# B&R Automation Studio project NAEUL004C00R13L518F00 (part 76)

#### Act_Main.st
```iecst
(** 2019-05-28 **)
ACTION Act_Main:

	IF eStatOld <> eStat THEN
		fbInit(bEn := FALSE);
		fbEnt(bEn := FALSE);
		fbPreExit(bEn := FALSE);
		fbExit(bEn := FALSE);
		fbExit1(bEn := FALSE);
		fbStop(bEn := FALSE);
		fbClprClampChk(bEn := FALSE);
		fbClprUnclampChk(bEn := FALSE);

		IF eStatOld <> MagConvActIdle
			AND eStatOld <> MagConvActSetMtrSigOnOrLToR
			AND eStatOld <> MagConvActSetMtrDirOrRToL
			AND eStatOld <> MagConvActRstMtrSigOnOrLToR
			AND eStatOld <> MagConvActRstMtrDirOrRToL
			AND eStatOld <> MagConvActSetMtrAll
			AND eStatOld <> MagConvActRstMtrAll THEN

			bMtrSigOnOrLToR	:= FALSE;
			bMtrDirOrRToL	:= FALSE;

		END_IF

		usiStep		:= 0;
		bReachEnd	:= FALSE;

		sStatTxt	:= a_sStatText[eStat];

		eStatOld	:= eStat;

		eStatus		:= Busy;
	END_IF

	//Main
	CASE eStat OF

		MagConvActIdle:
			IF EDGENEG(p_bManual) THEN
				bMtrSigOnOrLToR	:= FALSE;
				bMtrDirOrRToL	:= FALSE;
			END_IF

			eStatus	:= Idle;

		MagConvActInit:
			IF eStatus = Idle OR eStatus = Busy THEN

				eStatus	:= Busy;

				//Magazine Conveyor Init Run
				//Detect Have Magazine
				IF p_bLeftSen OR p_bRightSen THEN
					bHvMag	:= TRUE;
				ELSE
					bHvMag	:= FALSE;
				END_IF

				fbInit.bConvLToR	:= (p_eDirection = ConvDirLToR) OR (p_eDirection = ConvDirLToL);
				fbInit.tTxDlyTm		:= DINT_TO_TIME(p_diInitTm);

				IF fbInit.bConvLToR = TRUE THEN
					fbInit.bEndSen	:= p_bRightSen;
				ELSE
					fbInit.bEndSen	:= p_bLeftSen;
				END_IF

				fbInit(bEn := TRUE);

				bMtrSigOnOrLToR	:= fbInit.bMtrSigOnOrLToR;
				bMtrDirOrRToL	:= fbInit.bMtrDirOrRToL;

				IF fbInit.udiStatus = 0 THEN
					IF fbInit.bConvLToR = TRUE THEN
						IF bHvMag = TRUE AND p_bRightSen = FALSE THEN
							udiStatus	:= 10000;	//Magazine Detected But Not Present At Outlet Sensor (L - R) While Magazine Conveyor Initial
							eStatus		:= Error;
						ELSE
							eStatus	:= Done;
						END_IF
					ELSE
						IF bHvMag = TRUE AND p_bLeftSen = FALSE THEN
							udiStatus	:= 10001;	//Magazine Detected But Not Present At Outlet Sensor (R - L) While Magazine Conveyor Initial
							eStatus		:= Error;
						ELSE
							eStatus	:= Done;
						END_IF
					END_IF
				ELSIF fbInit.udiStatus < 65534 THEN
					udiStatus	:= fbInit.udiStatus;
					eStatus		:= Error;
				END_IF
			END_IF

		MagConvActInitStopClp:
			IF eStatus = Idle OR eStatus = Busy THEN

				eStatus	:= Busy;

				CASE usiStep OF
					0: //Unclamp
						bClprClampCtrl		:= FALSE;

						fbClprUnclampChk.bExtSen	:= p_bClprClampSen;
						fbClprUnclampChk.bRetSen	:= p_bClprUnclampSen;
						fbClprUnclampChk.bRetSafety	:= p_bClprUnclampSafetySen;
						fbClprUnclampChk(bEn := TRUE);

						IF fbClprUnclampChk.udiStatus = 0 THEN
							usiStep	:= 1;
						ELSIF fbClprUnclampChk.udiStatus < 65534 THEN
							bClprClampCtrl		:= TRUE;

							eStatus			:= Error;

							IF fbClprUnclampChk.udiStatus = 1504 THEN
								udiStatus	:= 10002;	//Clamper Clamp Sensor Off Time Out In Unclamp Check While Conveyor Initial With Clamper
							ELSIF fbClprUnclampChk.udiStatus = 1505 THEN
								udiStatus	:= 10003;	//Clamper Unclamp Sensor On Time Out In Unclamp Check While Conveyor Initial With Clamper
							ELSIF fbClprUnclampChk.udiStatus = 1508 THEN
								udiStatus	:= 10004;	//Clamper Unclamp Safety Sensor Error In Unclamp Check While Conveyor Initial With Clamper
							ELSE
								udiStatus	:= fbClprUnclampChk.udiStatus;
							END_IF
						END_IF

					1:	//Magazine Conveyor Init Run
						//Detect Have Magazine
						IF p_bLeftSen OR p_bRightSen THEN
							bHvMag	:= TRUE;
						ELSE
							bHvMag	:= FALSE;
						END_IF

						fbInit.bConvLToR	:= (p_eDirection = ConvDirLToR) OR (p_eDirection = ConvDirLToL);
						fbInit.tTxDlyTm		:= DINT_TO_TIME(p_diInitTm);

						IF fbInit.bConvLToR = TRUE THEN
							fbInit.bEndSen	:= p_bRightSen;
						ELSE
							fbInit.bEndSen	:= p_bLeftSen;
						END_IF

						fbInit(bEn := TRUE);

						bMtrSigOnOrLToR	:= fbInit.bMtrSigOnOrLToR;
						bMtrDirOrRToL	:= fbInit.bMtrDirOrRToL;

						IF fbInit.udiStatus = 0 THEN
							IF fbInit.bConvLToR = TRUE THEN
								IF bHvMag = TRUE AND p_bRightSen = FALSE THEN
									udiStatus	:= 10005;	//Magazine Detected But Not Present At Outlet Sensor (L - R) While Conveyor Initial With Clamper
									eStatus		:= Error;
								ELSE
									usiStep	:= 2;
								END_IF
							ELSE
								IF bHvMag = TRUE AND p_bLeftSen = FALSE THEN
									udiStatus	:= 10006;	//Magazine Detected But Not Present At Outlet Sensor (R - L) While Conveyor Initial With Clamper
									eStatus		:= Error;
								ELSE
									usiStep	:= 2;
								END_IF
							END_IF
						ELSIF fbInit.udiStatus < 65534 THEN
							udiStatus	:= fbInit.udiStatus;
							eStatus		:= Error;
						END_IF

					2:	//Check If Have Magazine
						IF bHvMag = TRUE THEN
							usiStep	:= 3;
						ELSE
							eStatus	:= Done;
						END_IF

					3:	//Clamp
						bClprClampCtrl		:= TRUE;

						fbClprClampChk.bExtSen		:= p_bClprClampSen;
						fbClprClampChk.bRetSen		:= p_bClprUnclampSen;
						fbClprClampChk.bExtSafety	:= p_bClprClampSafetySen;
						fbClprClampChk(bEn := TRUE);

						IF fbClprClampChk.udiStatus = 0 THEN
							eStatus		:= Done;
						ELSIF fbClprClampChk.udiStatus < 65534 THEN
							bClprClampCtrl		:= FALSE;

							eStatus			:= Error;

							IF fbClprClampChk.udiStatus = 1503 THEN
								udiStatus	:= 10007;	//Clamper Clamp Sensor On Time Out In Clamp Check While Conveyor Initial With Clamper
							ELSIF fbClprClampChk.udiStatus = 1506 THEN
								udiStatus	:= 10008;	//Clamper Unclamp Sensor Off Time Out In Clamp Check While Conveyor Initial With Clamper
							ELSIF fbClprClampChk.udiStatus = 1507 THEN
								udiStatus	:= 10009;	//Clamper Clamp Safety Sensor Error In Clamp Check While Conveyor Initial With Clamper
							ELSE
								udiStatus	:= fbClprClampChk.udiStatus;
							END_IF
						END_IF

				END_CASE
			END_IF

		MagConvActInitClpStop:
			IF eStatus = Idle OR eStatus = Busy THEN

				eStatus	:= Busy;

				CASE usiStep OF
					0: //Unclamp
						bClprClampCtrl		:= FALSE;

						fbClprUnclampChk.bExtSen	:= p_bClprClampSen;
						fbClprUnclampChk.bRetSen	:= p_bClprUnclampSen;
						fbClprUnclampChk.bRetSafety	:= p_bClprUnclampSafetySen;
						fbClprUnclampChk(bEn := TRUE);

						IF fbClprUnclampChk.udiStatus = 0 THEN
							usiStep	:= 1;
						ELSIF fbClprUnclampChk.udiStatus < 65534 THEN
							bClprClampCtrl		:= TRUE;

							eStatus			:= Error;

							IF fbClprUnclampChk.udiStatus = 1504 THEN
								udiStatus	:= 10038;	//Clamper Clamp Sensor Off Time Out In Unclamp Check While Conveyor Initial With Clamper
							ELSIF fbClprUnclampChk.udiStatus = 1505 THEN
								udiStatus	:= 10039;	//Clamper Unclamp Sensor On Time Out In Unclamp Check While Conveyor Initial With Clamper
							ELSIF fbClprUnclampChk.udiStatus = 1508 THEN
								udiStatus	:= 10040;	//Clamper Unclamp Safety Sensor Error In Unclamp Check While Conveyor Initial With Clamper
							ELSE
								udiStatus	:= fbClprUnclampChk.udiStatus;
							END_IF
						END_IF

					1:	//Magazine Conveyor Init Run & Clamp
						//Detect Have Magazine
						IF p_bLeftSen OR p_bRightSen THEN
							bHvMag	:= TRUE;
						ELSE
							bHvMag	:= FALSE;
						END_IF

						fbInit.bConvLToR	:= (p_eDirection = ConvDirLToR) OR (p_eDirection = ConvDirLToL);
						fbInit.tTxDlyTm		:= DINT_TO_TIME(p_diInitTm);

						IF fbInit.bConvLToR = TRUE THEN
							fbInit.bEndSen	:= p_bRightSen;
						ELSE
							fbInit.bEndSen	:= p_bLeftSen;
						END_IF

						fbInit(bEn := TRUE);

						bMtrSigOnOrLToR	:= fbInit.bMtrSigOnOrLToR;
						bMtrDirOrRToL	:= fbInit.bMtrDirOrRToL;

						IF fbInit.bEndSen = TRUE THEN
							bReachEnd	:= TRUE;
						END_IF

						IF bReachEnd = TRUE THEN
							fbClprDlyTm(IN := TRUE);

							IF fbClprDlyTm.Q = TRUE THEN
								bClprClampCtrl		:= TRUE;

								fbClprClampChk.bExtSen		:= p_bClprClampSen;
								fbClprClampChk.bRetSen		:= p_bClprUnclampSen;
								fbClprClampChk.bExtSafety	:= p_bClprClampSafetySen;
								fbClprClampChk(bEn := TRUE);
							END_IF

						END_IF

						IF (fbInit.udiStatus = 0) AND ((fbClprClampChk.udiStatus = 0) OR (bReachEnd = FALSE)) THEN
							IF fbInit.bConvLToR = TRUE THEN
								IF bHvMag = TRUE AND p_bRightSen = FALSE THEN
									udiStatus	:= 10041;	//Magazine Detected But Not Present At Outlet Sensor (L - R) While Conveyor Initial With Clamper
									eStatus		:= Error;
								ELSE
									eStatus		:= Done;
								END_IF
							ELSE
								IF bHvMag = TRUE AND p_bLeftSen = FALSE THEN
									udiStatus	:= 10042;	//Magazine Detected But Not Present At Outlet Sensor (R - L) While Conveyor Initial With Clamper
									eStatus		:= Error;
								ELSE
									eStatus		:= Done;
								END_IF
							END_IF

						ELSIF fbInit.udiStatus > 0 AND fbInit.udiStatus < 65534 THEN
							udiStatus	:= fbInit.udiStatus;
							eStatus		:= Error;

						ELSIF fbClprClampChk.udiStatus > 0 AND fbClprClampChk.udiStatus < 65534 THEN
							bClprClampCtrl		:= FALSE;

							eStatus			:= Error;

							IF fbClprClampChk.udiStatus = 1503 THEN
								udiStatus	:= 10043;	//Clamper Clamp Sensor On Time Out In Clamp Check While Conveyor Initial With Clamper
							ELSIF fbClprClampChk.udiStatus = 1506 THEN
								udiStatus	:= 10044;	//Clamper Unclamp Sensor Off Time Out In Clamp Check While Conveyor Initial With Clamper
							ELSIF fbClprClampChk.udiStatus = 1507 THEN
								udiStatus	:= 10045;	//Clamper Clamp Safety Sensor Error In Clamp Check While Conveyor Initial With Clamper
							ELSE
								udiStatus	:= fbClprClampChk.udiStatus;
							END_IF
						END_IF

				END_CASE
			END_IF

		MagConvActEnt:
			IF eStatus = Idle OR eStatus = Busy THEN

				eStatus	:= Busy;

				//Detect Have Magazine
				IF p_bLeftSen OR p_bRightSen THEN
					bHvMag	:= TRUE;
				END_IF

				//Conveyor Run
				fbEnt.bConvLToR		:= (p_eDirection = ConvDirLToR) OR (p_eDirection = ConvDirLToL);
				fbEnt.tTimeOut		:= DINT_TO_TIME(p_diTxInTimeOut);

				IF fbEnt.bConvLToR = TRUE THEN
					fbEnt.bEndSen	:= p_bRightSen;
				ELSE
					fbEnt.bEndSen	:= p_bLeftSen;
				END_IF

				fbEnt(bEn := TRUE);

				bMtrSigOnOrLToR	:= fbEnt.bMtrSigOnOrLToR;
				bMtrDirOrRToL	:= fbEnt.bMtrDirOrRToL;

				IF fbEnt.udiStatus = 0 THEN
					eStatus		:= Done;
				ELSIF fbEnt.udiStatus < 65534 THEN
					eStatus		:= Error;

					IF fbEnt.udiStatus = 1101 THEN
						udiStatus	:= 10028;	//Transfer In Time Out While Entering Magazine
					ELSE
						udiStatus	:= fbEnt.udiStatus;
					END_IF
				END_IF

			END_IF

		MagConvActEntStopClp:
			IF eStatus = Idle OR eStatus = Busy THEN

				eStatus	:= Busy;

				CASE usiStep OF
					0:
						//Detect Have Magazine
						IF p_bLeftSen OR p_bRightSen THEN
							bHvMag	:= TRUE;
						END_IF

						//Conveyor Run
						fbEnt.bConvLToR		:= (p_eDirection = ConvDirLToR) OR (p_eDirection = ConvDirLToL);
						fbEnt.tTimeOut		:= DINT_TO_TIME(p_diTxInTimeOut);

						IF fbEnt.bConvLToR = TRUE THEN
							fbEnt.bEndSen	:= p_bRightSen;
						ELSE
							fbEnt.bEndSen	:= p_bLeftSen;
						END_IF

						fbEnt(bEn := TRUE);

						bMtrSigOnOrLToR	:= fbEnt.bMtrSigOnOrLToR;
						bMtrDirOrRToL	:= fbEnt.bMtrDirOrRToL;

						IF fbEnt.udiStatus = 0 THEN
							usiStep	:= 1;
						ELSIF fbEnt.udiStatus < 65534 THEN
							eStatus		:= Error;

							IF fbEnt.udiStatus = 1101 THEN
								udiStatus	:= 10029;	//Transfer In Time Out While Entering Magazine
							ELSE
								udiStatus	:= fbEnt.udiStatus;
							END_IF
						END_IF

					1:
						bClprClampCtrl		:= TRUE;

						fbClprClampChk.bExtSen		:= p_bClprClampSen;
						fbClprClampChk.bRetSen		:= p_bClprUnclampSen;
						fbClprClampChk.bExtSafety	:= p_bClprClampSafetySen;
						fbClprClampChk(bEn := TRUE);

						IF fbClprClampChk.udiStatus = 0 THEN
							eStatus		:= Done;
						ELSIF fbClprClampChk.udiStatus < 65534 THEN
							bClprClampCtrl		:= FALSE;

							eStatus			:= Error;

							IF fbClprClampChk.udiStatus = 1503 THEN
								udiStatus	:= 10010;	//Clamper Clamp Sensor On Time Out In Clamp Check While Conveyor Enter With Clamper
							ELSIF fbClprClampChk.udiStatus = 1506 THEN
								udiStatus	:= 10011;	//Clamper Unclamp Sensor Off Time Out In Clamp Check While Conveyor Enter With Clamper
							ELSIF fbClprClampChk.udiStatus = 1507 THEN
								udiStatus	:= 10012;	//Clamper Clamp Safety Sensor Error In Clamp Check While Conveyor Enter With Clamper
							ELSE
								udiStatus	:= fbClprClampChk.udiStatus;
							END_IF
						END_IF

				END_CASE

			END_IF

		MagConvActEntClpStop:
			IF eStatus = Idle OR eStatus = Busy THEN

				eStatus	:= Busy;

				//Detect Have Magazine
				IF p_bLeftSen OR p_bRightSen THEN
					bHvMag	:= TRUE;
				END_IF

				//Conveyor Run
				fbEnt.bConvLToR		:= (p_eDirection = ConvDirLToR) OR (p_eDirection = ConvDirLToL);
				fbEnt.tTimeOut		:= DINT_TO_TIME(p_diTxInTimeOut);

				IF fbEnt.bConvLToR = TRUE THEN
					fbEnt.bEndSen	:= p_bRightSen;
				ELSE
					fbEnt.bEndSen	:= p_bLeftSen;
				END_IF

				fbEnt(bEn := TRUE);

				bMtrSigOnOrLToR	:= fbEnt.bMtrSigOnOrLToR;
				bMtrDirOrRToL	:= fbEnt.bMtrDirOrRToL;

				IF fbEnt.bEndSen = TRUE THEN
					bReachEnd	:= TRUE;
				END_IF

				IF bReachEnd = TRUE THEN
					fbClprDlyTm(IN := TRUE);

					IF fbClprDlyTm.Q = TRUE THEN
						bClprClampCtrl		:= TRUE;

						fbClprClampChk.bExtSen		:= p_bClprClampSen;
						fbClprClampChk.bRetSen		:= p_bClprUnclampSen;
						fbClprClampChk.bExtSafety	:= p_bClprClampSafetySen;
						fbClprClampChk(bEn := TRUE);
					END_IF

				END_IF

				IF fbClprClampChk.udiStatus = 0 AND fbEnt.udiStatus = 0 THEN
					eStatus		:= Done;

				ELSIF fbClprClampChk.udiStatus > 0 AND fbClprClampChk.udiStatus < 65534 THEN
					bClprClampCtrl		:= FALSE;

					eStatus			:= Error;

					IF fbClprClampChk.udiStatus = 1503 THEN
						udiStatus	:= 10034;	//Clamper Clamp Sensor On Time Out In Clamp Check While Conveyor Enter With Clamper
					ELSIF fbClprClampChk.udiStatus = 1506 THEN
						udiStatus	:= 10035;	//Clamper Unclamp Sensor Off Time Out In Clamp Check While Conveyor Enter With Clamper
					ELSIF fbClprClampChk.udiStatus = 1507 THEN
						udiStatus	:= 10036;	//Clamper Clamp Safety Sensor Error In Clamp Check While Conveyor Enter With Clamper
					ELSE
						udiStatus	:= fbClprClampChk.udiStatus;
					END_IF

				ELSIF fbEnt.udiStatus > 0 AND fbEnt.udiStatus < 65534 THEN
					eStatus		:= Error;

					IF fbEnt.udiStatus = 1101 THEN
						udiStatus	:= 10037;	//Transfer In Time Out While Entering Magazine
					ELSE
						udiStatus	:= fbEnt.udiStatus;
					END_IF

				END_IF

			END_IF

		MagConvActPreExit:
			IF eStatus = Idle OR eStatus = Busy THEN

				eStatus	:= Busy;

				//Conveyor Run
				fbPreExit.bConvLToR		:= (p_eDirection = ConvDirLToR) OR (p_eDirection = ConvDirRToR);
				fbPreExit.tTxDlyTm		:= DINT_TO_TIME(p_diInitTm);

				IF fbPreExit.bConvLToR = TRUE THEN
					fbPreExit.bEndSen	:= p_bRightSen;
				ELSE
					fbPreExit.bEndSen	:= p_bLeftSen;
				END_IF

				fbPreExit(bEn := TRUE);

				bMtrSigOnOrLToR	:= fbPreExit.bMtrSigOnOrLToR;
				bMtrDirOrRToL	:= fbPreExit.bMtrDirOrRToL;

				IF fbPreExit.udiStatus = 0 THEN
					IF fbPreExit.bEndSen = TRUE THEN
						eStatus	:= Done;
					ELSE
						udiStatus	:= 10046;	//Magazine Not Detected While Pre-Exiting Magazine
						eStatus		:= Error;
					END_IF
				ELSIF fbPreExit.udiStatus < 65534 THEN
					udiStatus	:= fbPreExit.udiStatus;
					eStatus		:= Error;
				END_IF

			END_IF

		MagConvActPreExitClpr:
			IF eStatus = Idle OR eStatus = Busy THEN

				eStatus	:= Busy;

				CASE usiStep OF
					0:
						bClprClampCtrl		:= FALSE;

						fbClprUnclampChk.bExtSen		:= p_bClprClampSen;
						fbClprUnclampChk.bRetSen		:= p_bClprUnclampSen;
						fbClprUnclampChk.bRetSafety		:= p_bClprUnclampSafetySen;
						fbClprUnclampChk(bEn := TRUE);

						IF fbClprUnclampChk.udiStatus = 0 THEN
							usiStep		:= 1;
						ELSIF fbClprUnclampChk.udiStatus < 65534 THEN
							bClprClampCtrl		:= TRUE;

							eStatus			:= Error;

							IF fbClprUnclampChk.udiStatus = 1504 THEN
								udiStatus	:= 10013;	//Clamper Clamp Sensor Off Time Out In Unclamp Check While Conveyor Exit With Clamper
							ELSIF fbClprUnclampChk.udiStatus = 1505 THEN
								udiStatus	:= 10014;	//Clamper Unclamp Sensor On Time Out In Unclamp Check While Conveyor Exit With Clamper
							ELSIF fbClprUnclampChk.udiStatus = 1508 THEN
								udiStatus	:= 10015;	//Clamper Unclamp Safety Sensor Error In Unclamp Check While Conveyor Exit With Clamper
							ELSE
								udiStatus	:= fbClprUnclampChk.udiStatus;
							END_IF
						END_IF

					1:
						//Conveyor Run
						fbPreExit.bConvLToR		:= (p_eDirection = ConvDirLToR) OR (p_eDirection = ConvDirRToR);
						fbPreExit.tTxDlyTm		:= DINT_TO_TIME(p_diInitTm);

						IF fbPreExit.bConvLToR = TRUE THEN
							fbPreExit.bEndSen	:= p_bRightSen;
						ELSE
							fbPreExit.bEndSen	:= p_bLeftSen;
						END_IF

						fbPreExit(bEn := TRUE);

						bMtrSigOnOrLToR	:= fbPreExit.bMtrSigOnOrLToR;
						bMtrDirOrRToL	:= fbPreExit.bMtrDirOrRToL;

						IF fbPreExit.udiStatus = 0 THEN
							IF fbPreExit.bEndSen = TRUE THEN
								eStatus	:= Done;
							ELSE
								udiStatus	:= 10046;	//Magazine Not Detected While Pre-Exiting Magazine
								eStatus		:= Error;
							END_IF
						ELSIF fbPreExit.udiStatus < 65534 THEN
							udiStatus	:= fbPreExit.udiStatus;
							eStatus		:= Error;
						END_IF

				END_CASE

			END_IF

		MagConvActExit:
			IF eStatus = Idle OR eStatus = Busy THEN

				eStatus	:= Busy;

				//Conveyor Run
				fbExit.bConvLToR	:= (p_eDirection = ConvDirLToR) OR (p_eDirection = ConvDirRToR);
				fbExit.tTimeOut		:= DINT_TO_TIME(p_diTxOutTimeOut);

				IF fbExit.bConvLToR = TRUE THEN
					fbExit.bEndSen	:= p_bRightSen;
				ELSE
					fbExit.bEndSen	:= p_bLeftSen;
				END_IF

				fbExit(bEn := TRUE);

				bMtrSigOnOrLToR	:= fbExit.bMtrSigOnOrLToR;
				bMtrDirOrRToL	:= fbExit.bMtrDirOrRToL;

				IF fbExit.udiStatus = 0 THEN
					bHvMag		:= FALSE;
					eStatus		:= Done;
				ELSIF fbExit.udiStatus < 65534 THEN
					eStatus		:= Error;

					IF fbExit.udiStatus = 1101 THEN
						udiStatus	:= 10030;	//Transfer Out Time Out While Exiting Magazine
					ELSE
						udiStatus	:= fbExit.udiStatus;
					END_IF
				END_IF

			END_IF

		MagConvActExit1:
			IF eStatus = Idle OR eStatus = Busy THEN

				eStatus	:= Busy;

				//Conveyor Run
				fbExit1.bConvLToR		:= (p_eDirection = ConvDirLToR) OR (p_eDirection = ConvDirRToR);
				fbExit1.tTimeOut		:= DINT_TO_TIME(p_diTxOutTimeOut);

				IF fbExit1.bConvLToR = TRUE THEN
					fbExit1.bEndSen	:= p_bRightSen;
				ELSE
					fbExit1.bEndSen	:= p_bLeftSen;
				END_IF

				fbExit1(bEn := TRUE);

				bMtrSigOnOrLToR	:= fbExit1.bMtrSigOnOrLToR;
				bMtrDirOrRToL	:= fbExit1.bMtrDirOrRToL;

				IF fbExit1.udiStatus = 0 THEN
					bHvMag		:= FALSE;
					eStatus		:= Done;
				ELSIF fbExit1.udiStatus < 65534 THEN
					eStatus		:= Error;

					IF fbExit1.udiStatus = 1101 THEN
						udiStatus	:= 10032;	//Transfer Out Time Out While Exiting Magazinie
					ELSE
						udiStatus	:= fbExit1.udiStatus;
					END_IF
				END_IF

			END_IF

		MagConvActExitClpr:
			IF eStatus = Idle OR eStatus = Busy THEN

				eStatus	:= Busy;

				CASE usiStep OF
					0:
						bClprClampCtrl		:= FALSE;

						fbClprUnclampChk.bExtSen		:= p_bClprClampSen;
						fbClprUnclampChk.bRetSen		:= p_bClprUnclampSen;
						fbClprUnclampChk.bRetSafety		:= p_bClprUnclampSafetySen;
						fbClprUnclampChk(bEn := TRUE);

						IF fbClprUnclampChk.udiStatus = 0 THEN
							usiStep		:= 1;
						ELSIF fbClprUnclampChk.udiStatus < 65534 THEN
							bClprClampCtrl		:= TRUE;

							eStatus			:= Error;

							IF fbClprUnclampChk.udiStatus = 1504 THEN
								udiStatus	:= 10013;	//Clamper Clamp Sensor Off Time Out In Unclamp Check While Conveyor Exit With Clamper
							ELSIF fbClprUnclampChk.udiStatus = 1505 THEN
								udiStatus	:= 10014;	//Clamper Unclamp Sensor On Time Out In Unclamp Check While Conveyor Exit With Clamper
							ELSIF fbClprUnclampChk.udiStatus = 1508 THEN
								udiStatus	:= 10015;	//Clamper Unclamp Safety Sensor Error In Unclamp Check While Conveyor Exit With Clamper
							ELSE
								udiStatus	:= fbClprUnclampChk.udiStatus;
							END_IF
						END_IF

					1:
						//Conveyor Run
						fbExit.bConvLToR	:= (p_eDirection = ConvDirLToR) OR (p_eDirection = ConvDirRToR);
						fbExit.tTimeOut		:= DINT_TO_TIME(p_diTxOutTimeOut);

						IF fbExit.bConvLToR = TRUE THEN
							fbExit.bEndSen	:= p_bRightSen;
						ELSE
							fbExit.bEndSen	:= p_bLeftSen;
						END_IF

						fbExit(bEn := TRUE);

						bMtrSigOnOrLToR	:= fbExit.bMtrSigOnOrLToR;
						bMtrDirOrRToL	:= fbExit.bMtrDirOrRToL;

						IF fbExit.udiStatus = 0 THEN
							bHvMag		:= FALSE;
							eStatus		:= Done;
						ELSIF fbExit.udiStatus < 65534 THEN
							eStatus		:= Error;

							IF fbExit.udiStatus = 1101 THEN
								udiStatus	:= 10031;	//Transfer Out Time Out While Conveyor Exit With Clamper
							ELSE
								udiStatus	:= fbExit.udiStatus;
							END_IF
						END_IF

				END_CASE

			END_IF

		MagConvActExit1Clpr:
			IF eStatus = Idle OR eStatus = Busy THEN

				eStatus	:= Busy;

				CASE usiStep OF
					0:
						bClprClampCtrl		:= FALSE;

						fbClprUnclampChk.bExtSen		:= p_bClprClampSen;
						fbClprUnclampChk.bRetSen		:= p_bClprUnclampSen;
						fbClprUnclampChk.bRetSafety		:= p_bClprUnclampSafetySen;
						fbClprUnclampChk(bEn := TRUE);

						IF fbClprUnclampChk.udiStatus = 0 THEN
							usiStep		:= 1;
						ELSIF fbClprUnclampChk.udiStatus < 65534 THEN
							bClprClampCtrl		:= TRUE;

							eStatus			:= Error;

							IF fbClprUnclampChk.udiStatus = 1504 THEN
								udiStatus	:= 10025;	//Clamper Clamp Sensor Off Time Out In Unclamp Check While Conveyor Exit With Clamper
							ELSIF fbClprUnclampChk.udiStatus = 1505 THEN
								udiStatus	:= 10026;	//Clamper Unclamp Sensor On Time Out In Unclamp Check While Conveyor Exit With Clamper
							ELSIF fbClprUnclampChk.udiStatus = 1508 THEN
								udiStatus	:= 10027;	//Clamper Unclamp Safety Sensor Error In Unclamp Check While Conveyor Exit With Clamper
							ELSE
								udiStatus	:= fbClprUnclampChk.udiStatus;
							END_IF
						END_IF

					1:
						//Conveyor Run
						fbExit1.bConvLToR		:= (p_eDirection = ConvDirLToR) OR (p_eDirection = ConvDirRToR);
						fbExit1.tTimeOut		:= DINT_TO_TIME(p_diTxOutTimeOut);

						IF fbExit1.bConvLToR = TRUE THEN
							fbExit1.bEndSen	:= p_bRightSen;
						ELSE
							fbExit1.bEndSen	:= p_bLeftSen;
						END_IF

						fbExit1(bEn := TRUE);

						bMtrSigOnOrLToR	:= fbExit1.bMtrSigOnOrLToR;
						bMtrDirOrRToL	:= fbExit1.bMtrDirOrRToL;

						IF fbExit1.udiStatus = 0 THEN
							bHvMag		:= FALSE;
							eStatus		:= Done;
						ELSIF fbExit1.udiStatus < 65534 THEN
							eStatus		:= Error;

							IF fbExit1.udiStatus = 1101 THEN
								udiStatus	:= 10033;	//Transfer Out Time Out While Conveyor Exit With Clamper
							ELSE
								udiStatus	:= fbExit1.udiStatus;
							END_IF
						END_IF

				END_CASE

			END_IF

		MagConvActClprSetAll:
			IF eStatus = Idle OR eStatus = Busy THEN

				eStatus	:= Busy;

				bMtrSigOnOrLToR	:= FALSE;
				bMtrDirOrRToL	:= FALSE;

				bClprClampCtrl		:= TRUE;

				eStatus		:= Done;

			END_IF

		MagConvActClprRstAll:
			IF eStatus = Idle OR eStatus = Busy THEN

				eStatus	:= Busy;

				bMtrSigOnOrLToR	:= FALSE;
				bMtrDirOrRToL	:= FALSE;

				bClprClampCtrl		:= FALSE;

				eStatus		:= Done;

			END_IF

		MagConvActClprSetClamp:
			IF eStatus = Idle OR eStatus = Busy THEN

				eStatus	:= Busy;

				bMtrSigOnOrLToR	:= FALSE;
				bMtrDirOrRToL	:= FALSE;

				bClprClampCtrl		:= TRUE;

				eStatus		:= Done;

			END_IF

		MagConvActClprSetUnclamp:
			IF eStatus = Idle OR eStatus = Busy THEN

				eStatus	:= Busy;

				bMtrSigOnOrLToR	:= FALSE;
				bMtrDirOrRToL	:= FALSE;

				bClprClampCtrl		:= FALSE;

				eStatus		:= Done;

			END_IF

		MagConvActClprClamp:
			IF eStatus = Idle OR eStatus = Busy THEN

				eStatus	:= Busy;

				bMtrSigOnOrLToR	:= FALSE;
				bMtrDirOrRToL	:= FALSE;

				bClprClampCtrl		:= TRUE;

				fbClprClampChk.bExtSen		:= p_bClprClampSen;
				fbClprClampChk.bRetSen		:= p_bClprUnclampSen;
				fbClprClampChk.bExtSafety	:= p_bClprClampSafetySen;
				fbClprClampChk(bEn := TRUE);

				IF fbClprClampChk.udiStatus = 0 THEN
					eStatus		:= Done;
				ELSIF fbClprClampChk.udiStatus < 65534 THEN
					bClprClampCtrl		:= FALSE;

					eStatus			:= Error;

					IF fbClprClampChk.udiStatus = 1503 THEN
						udiStatus	:= 10016;	//Clamper Clamp Sensor On Time Out In Clamp Check While Clamper Clamp
					ELSIF fbClprClampChk.udiStatus = 1506 THEN
						udiStatus	:= 10017;	//Clamper Unclamp Sensor Off Time Out In Clamp Check While Clamper Clamp
					ELSIF fbClprClampChk.udiStatus = 1507 THEN
						udiStatus	:= 10018;	//Clamper Clamp Safety Sensor Error In Clamp Check While Clamper Clamp
					ELSE
						udiStatus	:= fbClprClampChk.udiStatus;
					END_IF
				END_IF
			END_IF

		MagConvActClprUnclamp:
			IF eStatus = Idle OR eStatus = Busy THEN

				eStatus	:= Busy;

				bMtrSigOnOrLToR	:= FALSE;
				bMtrDirOrRToL	:= FALSE;

				bClprClampCtrl		:= FALSE;

				fbClprUnclampChk.bExtSen		:= p_bClprClampSen;
				fbClprUnclampChk.bRetSen		:= p_bClprUnclampSen;
				fbClprUnclampChk.bRetSafety		:= p_bClprUnclampSafetySen;
				fbClprUnclampChk(bEn := TRUE);

				IF fbClprUnclampChk.udiStatus = 0 THEN
					eStatus		:= Done;
				ELSIF fbClprUnclampChk.udiStatus < 65534 THEN
					bClprClampCtrl		:= TRUE;

					eStatus			:= Error;

					IF fbClprUnclampChk.udiStatus = 1504 THEN
						udiStatus	:= 10019;	//Clamper Clamp Sensor Off Time Out In Unclamp Check While Clamper Unclamp
					ELSIF fbClprUnclampChk.udiStatus = 1505 THEN
						udiStatus	:= 10020;	//Clamper Unclamp Sensor On Time Out In Unclamp Check While Clamper Unclamp
					ELSIF fbClprUnclampChk.udiStatus = 1508 THEN
						udiStatus	:= 10021;	//Clamper Unclamp Safety Sensor Error In Unclamp Check While Clamper Unclamp
					ELSE
						udiStatus	:= fbClprUnclampChk.udiStatus;
					END_IF
				END_IF

			END_IF

		MagConvActStop:
			IF eStatus = Idle OR eStatus = Busy THEN

				eStatus	:= Busy;

				//Conveyor Run
				fbStop(bEn := TRUE);

				bMtrSigOnOrLToR	:= fbStop.bMtrSigOnOrLToR;
				bMtrDirOrRToL	:= fbStop.bMtrDirOrRToL;

				IF fbStop.udiStatus = 0 THEN
					eStatus	:= Done;
				ELSIF fbStop.udiStatus < 65534 THEN
					udiStatus	:= fbStop.udiStatus;
					eStatus		:= Error;
				END_IF

			END_IF

		MagConvActStopClpr:
			IF eStatus = Idle OR eStatus = Busy THEN

				eStatus	:= Busy;

				//Conveyor Run
				fbStop(bEn := TRUE);

				bMtrSigOnOrLToR	:= fbStop.bMtrSigOnOrLToR;
				bMtrDirOrRToL	:= fbStop.bMtrDirOrRToL;

				bClprClampCtrl		:= FALSE;

				fbClprUnclampChk.bExtSen		:= p_bClprClampSen;
				fbClprUnclampChk.bRetSen		:= p_bClprUnclampSen;
				fbClprUnclampChk.bRetSafety		:= p_bClprUnclampSafetySen;
				fbClprUnclampChk(bEn := TRUE);

				IF fbStop.udiStatus = 0 AND fbClprUnclampChk.udiStatus = 0 THEN
					eStatus		:= Done;
				ELSIF fbStop.udiStatus > 0 AND fbStop.udiStatus < 65534 THEN
					udiStatus	:= fbStop.udiStatus;
					eStatus		:= Error;
				ELSIF fbClprUnclampChk.udiStatus > 0 AND fbClprUnclampChk.udiStatus < 65534 THEN
					bClprClampCtrl		:= TRUE;

					eStatus			:= Error;

					IF fbClprUnclampChk.udiStatus = 1504 THEN
						udiStatus	:= 10022;	//Clamper Clamp Sensor Off Time Out In Unclamp Check While Stop With Clamper
					ELSIF fbClprUnclampChk.udiStatus = 1505 THEN
						udiStatus	:= 10023;	//Clamper Unclamp Sensor On Time Out In Unclamp Check While Stop With Clamper
					ELSIF fbClprUnclampChk.udiStatus = 1508 THEN
						udiStatus	:= 10024;	//Clamper Unclamp Safety Sensor Error In Unclamp Check While Stop With Clamper
					ELSE
						udiStatus	:= fbClprUnclampChk.udiStatus;
					END_IF
				END_IF

			END_IF

		MagConvActSetMtrSigOnOrLToR:
			IF eStatus = Idle OR eStatus = Busy THEN

				bMtrSigOnOrLToR	:= TRUE;

				eStatus		:= Done;

			END_IF

		MagConvActSetMtrDirOrRToL:
			IF eStatus = Idle OR eStatus = Busy THEN

				bMtrDirOrRToL	:= TRUE;

				eStatus		:= Done;

			END_IF

		MagConvActRstMtrSigOnOrLToR:
			IF eStatus = Idle OR eStatus = Busy THEN

				bMtrSigOnOrLToR	:= FALSE;

				eStatus		:= Done;

			END_IF

		MagConvActRstMtrDirOrRToL:
			IF eStatus = Idle OR eStatus = Busy THEN

				bMtrDirOrRToL	:= FALSE;

				eStatus		:= Done;

			END_IF

		MagConvActSetMtrAll:
			IF eStatus = Idle OR eStatus = Busy THEN

				bMtrSigOnOrLToR	:= TRUE;
				bMtrDirOrRToL	:= TRUE;

				eStatus		:= Done;

			END_IF

		MagConvActRstMtrAll:
			IF eStatus = Idle OR eStatus = Busy THEN

				bMtrSigOnOrLToR	:= FALSE;
				bMtrDirOrRToL	:= FALSE;

				eStatus		:= Done;

			END_IF

	END_CASE

END_ACTION
```

#### Init.st
```iecst
(** 2019-03-25 **)
PROGRAM _INIT

	(* Always Change If Project Change *)

	//Pass Address To Global Address For External Use
	//Action, State & Status
	p_OutMagConvStat		:= ADR(eStat);
	p_OutMagConvStatus		:= ADR(eStatus);
	p_OutMagConvStatTxt		:= ADR(sStatTxt);

	//Alarm
	p_OutMagConvAlmData		:= ADR(tyAlmData);

	//Output
	p_OutMagConvHvMag					:= ADR(bHvMag);
	p_OutMagConvMtrSigOnOrLToR			:= ADR(bMtrSigOnOrLToR);
	p_OutMagConvMtrDirOrRToL			:= ADR(bMtrDirOrRToL);

	p_OutMagConvClprClampCtrl			:= ADR(bClprClampCtrl);
	p_OutMagConvClprTwoOutControl		:= ADR(bClprTwoOutputControl);

	(* Always Change If Project Change *)

END_PROGRAM
```

### LifterMagConv.var - Change By Project
```iecst
(*2019-03-25*)
(**)
(*Action & State & Status*)
VAR
	p_LifterMagConvStat : UDINT;
	p_LifterMagConvStatus : UDINT;
	p_LifterMagConvStatTxt : UDINT;
END_VAR
(**)
(*Alarm*)
VAR
	p_LifterMagConvAlmData : UDINT;
END_VAR
(**)
(*Output*)
VAR
	p_LifterMagConvHvMag : UDINT;
	p_LifterMagConvMtrSigOnOrLToR : UDINT;
	p_LifterMagConvMtrDirOrRToL : UDINT;
	p_LifterMagConvClprClampCtrl : UDINT;
	p_LifterMagConvClprTwoOutputCtrl : UDINT;
END_VAR
```

### Program Logical/MagConv_TopBtm/LifterMagConv (IEC) - 1.00.0 - NtConv v5.00.0 , NtPneu v5.00.0

#### InputRef.var
```iecst
(*2019-03-25*)
(**)
(*General*)
VAR
	p_eAct : REFERENCE TO eMagConvAction;
	p_udiRstErr : REFERENCE TO UDINT;
	p_bPrep : REFERENCE TO BOOL;
	p_bEn : REFERENCE TO BOOL;
	p_bDis : REFERENCE TO BOOL;
END_VAR
(**)
(*Configuration*)
VAR
	p_bManual : REFERENCE TO BOOL;
	p_bOnDirMod : REFERENCE TO BOOL;
	p_diInitTm : REFERENCE TO DINT;
	p_tMtrOffDlyTm : REFERENCE TO TIME;
	p_diTxInTimeOut : REFERENCE TO DINT;
	p_diTxOutTimeOut : REFERENCE TO DINT;
	p_eDirection : REFERENCE TO eConvDir;
	p_sProgNm : REFERENCE TO STRING[15];
	p_tClprClampTO : REFERENCE TO TIME;
	p_tClprUnclampTO : REFERENCE TO TIME;
	p_bNtSettingsLoadDone : REFERENCE TO BOOL;
END_VAR
(**)
(*Input*)
VAR
	p_bLeftSen : REFERENCE TO BOOL;
	p_bRightSen : REFERENCE TO BOOL;
	p_bClprClampSen : REFERENCE TO BOOL;
	p_bClprUnclampSen : REFERENCE TO BOOL;
	p_bClprClampSafetySen : REFERENCE TO BOOL;
	p_bClprUnclampSafetySen : REFERENCE TO BOOL;
	p_bMagPresentSen : REFERENCE TO BOOL;
END_VAR
```

#### InputRef_Link.var
```iecst
(*2019-04-09*)
(**)
(*External*)
VAR
	p_bLinkOpsRun : REFERENCE TO BOOL;
END_VAR
(**)
VAR
	p_bLinkDISafetyRlySig : REFERENCE TO BOOL;
	p_diLinkLifterActualPos : REFERENCE TO DINT;
	p_diLinkLifterBtmPos : REFERENCE TO DINT;
	p_diLinkLifterTopPos : REFERENCE TO DINT;
	p_bLinkOpsInitULDStepInitDone : REFERENCE TO BOOL;
	p_bLinkTopMagConvEntSen : REFERENCE TO BOOL;
	p_bLinkOpsLifMagULStepExtMag1 : REFERENCE TO BOOL;
END_VAR
(**)
VAR
	fbLeftSenOnChk : TON;
	fbLeftSenOn : TON;
END_VAR
```

#### Local.var
```iecst
(*2019-05-28*)
(**)
(*Local Action, State & Status*)
VAR
	eAct : eMagConvAction := MagConvActIdle;
	eStat : eMagConvAction := MagConvActIdle;
	eStatus : eFBStatus := Idle;
	udiStatus : UDINT := 0;
	sStatTxt : STRING[200] := '';
	a_sStatText : ARRAY[0..50] OF STRING[200] := ['Idling','Initializing','Initializing With Stop Then Clamper','Initializing With Clamper Then Stop','Entering Board','Entering Board With Stop Then Clamper','Entering Board With Clamper Then Stop',2('Exiting Board'),2('Exiting Board With Clamper'),'Clamper Setting All Control','Clamper Resetting All Control','Clamper Setting Clamp','Clamper Setting Unclamp','Clamper Clamp','Clampler Unclamp','Stopping','Stopping With Clamper','Turning On Motor Signal','Turning On Motor Direction','Turning Off Motor Signal','Turning Off Motor Direction','Turning On All Motor Output','Turning Off All Motor Output',26('')];
END_VAR
(**)
(*Local Alarm*)
VAR
	tyAlmData : tyAlmDat;
	a_tyAlmText : ARRAY[10000..10099] OF tyAlmTxt := [(sAlmText:='Magazine Detected But Not Present At Outlet Sensor (L - R) While Magazine Conveyor Initial',sRcyText:='Operation Interrupted By Undetected Magazine. Adjusting The Magazine Or Remove The Present Magazine To Resume Operation.'),(sAlmText:='Magazine Detected But Not Present At Outlet Sensor (R - L) While Magazine Conveyor Initial',sRcyText:='Operation Interrupted By Undetected Magazine. Adjusting The Magazine Or Remove The Present Magazine To Resume Operation.'),(sAlmText:='Clamper Clamp Sensor Off Time Out In Unclamp Check While Conveyor Initial With Clamper',sRcyText:='Sensor Timeout Expired Before Operation Completed. Sensor Operation Is Abnormal. Solve The Error To Resume Operation.'),(sAlmText:='Clamper Unclamp Sensor On Time Out In Unclamp Check While Conveyor Initial With Clamper',sRcyText:='Sensor Timeout Expired Before Operation Completed. Sensor Operation Is Abnormal. Solve The Error To Resume Operation.'),(sAlmText:='Clamper Unclamp Safety Sensor Error In Unclamp Check While Conveyor Initial With Clamper',sRcyText:='Safety System Has Been Triggered. All Operations Are Disable. Remove the Obstacle That Triggered The Safety Interlock To Resume Operation.'),(sAlmText:='Magazine Detected But Not Present At Outlet Sensor (L - R) While Conveyor Initial With Clamper',sRcyText:='Operation Interrupted By Undetected Magazine. Adjusting The Magazine Or Remove The Present Magazine To Resume Operation.'),(sAlmText:='Magazine Detected But Not Present At Outlet Sensor (R - L) While Conveyor Initial With Clamper',sRcyText:='Operation Interrupted By Undetected Magazine. Adjusting The Magazine Or Remove The Present Magazine To Resume Operation.'),(sAlmText:='Clamper Clamp Sensor On Time Out In Clamp Check While Conveyor Initial With Clamper',sRcyText:='Sensor Timeout Expired Before Operation Completed. Sensor Operation Is Abnormal. Solve The Error To Resume Operation.'),(sAlmText:='Clamper Unclamp Sensor Off Time Out In Clamp Check While Conveyor Initial With Clamper',sRcyText:='Sensor Timeout Expired Before Operation Completed. Sensor Operation Is Abnormal. Solve The Error To Resume Operation.'),(sAlmText:='Clamper Clamp Safety Sensor Error In Clamp Check While Conveyor Initial With Clamper',sRcyText:='Safety System Has Been Triggered. All Operations Are Disable. Remove the Obstacle That Triggered The Safety Interlock To Resume Operation.'),(sAlmText:='Clamper Clamp Sensor On Time Out In Clamp Check While Conveyor Enter With Clamper',sRcyText:='Sensor Timeout Expired Before Operation Completed. Sensor Operation Is Abnormal. Solve The Error To Resume Operation.'),(sAlmText:='Clamper Unclamp Sensor Off Time Out In Clamp Check While Conveyor Enter With Clamper',sRcyText:='Sensor Timeout Expired Before Operation Completed. Sensor Operation Is Abnormal. Solve The Error To Resume Operation.'),(sAlmText:='Clamper Clamp Safety Sensor Error In Clamp Check While Conveyor Enter With Clamper',sRcyText:='Safety System Has Been Triggered. All Operations Are Disable. Remove the Obstacle That Triggered The Safety Interlock To Resume Operation.'),(sAlmText:='Clamper Clamp Sensor Off Time Out In Unclamp Check While Conveyor Exit With Clamper',sRcyText:='Sensor Timeout Expired Before Operation Completed. Sensor Operation Is Abnormal. Solve The Error To Resume Operation.'),(sAlmText:='Clamper Unclamp Sensor On Time Out In Unclamp Check While Conveyor Exit With Clamper',sRcyText:='Sensor Timeout Expired Before Operation Completed. Sensor Operation Is Abnormal. Solve The Error To Resume Operation.'),(sAlmText:='Clamper Unclamp Safety Sensor Error In Unclamp Check While Conveyor Exit With Clamper',sRcyText:='Safety System Has Been Triggered. All Operations Are Disable. Remove the Obstacle That Triggered The Safety Interlock To Resume Operation.'),(sAlmText:='Clamper Clamp Sensor On Time Out In Clamp Check While Clamper Clamp',sRcyText:='Sensor Timeout Expired Before Operation Completed. Sensor Operation Is Abnormal. Solve The Error To Resume Operation.'),(sAlmText:='Clamper Unclamp Sensor Off Time Out In Clamp Check While Clamper Clamp',sRcyText:='Sensor Timeout Expired Before Operation Completed. Sensor Operation Is Abnormal. Solve The Error To Resume Operation.'),(sAlmText:='Clamper Clamp Safety Sensor Error In Clamp Check While Clamper Clamp',sRcyText:='Safety System Has Been Triggered. All Operations Are Disable. Remove the Obstacle That Triggered The Safety Interlock To Resume Operation.'),(sAlmText:='Clamper Clamp Sensor Off Time Out In Unclamp Check While Clamper Unclamp',sRcyText:='Sensor Timeout Expired Before Operation Completed. Sensor Operation Is Abnormal. Solve The Error To Resume Operation.'),(sAlmText:='Clamper Unclamp Sensor On Time Out In Unclamp Check While Clamper Unclamp',sRcyText:='Sensor Timeout Expired Before Operation Completed. Sensor Operation Is Abnormal. Solve The Error To Resume Operation.'),(sAlmText:='Clamper Unclamp Safety Sensor Error In Unclamp Check While Clamper Unclamp',sRcyText:='Safety System Has Been Triggered. All Operations Are Disable. Remove the Obstacle That Triggered The Safety Interlock To Resume Operation.'),(sAlmText:='Clamper Clamp Sensor Off Time Out In Unclamp Check While Stop With Clamper',sRcyText:='Sensor Timeout Expired Before Operation Completed. Sensor Operation Is Abnormal. Solve The Error To Resume Operation.'),(sAlmText:='Clamper Unclamp Sensor On Time Out In Unclamp Check While Stop With Clamper',sRcyText:='Sensor Timeout Expired Before Operation Completed. Sensor Operation Is Abnormal. Solve The Error To Resume Operation.'),(sAlmText:='Clamper Unclamp Safety Sensor Error In Unclamp Check While Stop With Clamper',sRcyText:='Safety System Has Been Triggered. All Operations Are Disable. Remove the Obstacle That Triggered The Safety Interlock To Resume Operation.'),(sAlmText:='Clamper Clamp Sensor Off Time Out In Unclamp Check While Conveyor Exit With Clamper',sRcyText:='Sensor Timeout Expired Before Operation Completed. Sensor Operation Is Abnormal. Solve The Error To Resume Operation.'),(sAlmText:='Clamper Unclamp Sensor On Time Out In Unclamp Check While Conveyor Exit With Clamper',sRcyText:='Sensor Timeout Expired Before Operation Completed. Sensor Operation Is Abnormal. Solve The Error To Resume Operation.'),(sAlmText:='Clamper Unclamp Safety Sensor Error In Unclamp Check While Conveyor Exit With Clamper',sRcyText:='Safety System Has Been Triggered. All Operations Are Disable. Remove the Obstacle That Triggered The Safety Interlock To Resume Operation.'),2((sAlmText:='Transfer In Time Out While Entering Magazine',sRcyText:='Timeout Expired Before Operation Completed. Transmission Abnormal. Remove the Obstacle (If Exists) To Resume Operation.')),(sAlmText:='Transfer Out Time Out While Exiting Magazine',sRcyText:='Timeout Expired Before Operation Completed. Transmission Abnormal. Remove the Obstacle (If Exists) To Resume Operation.'),(sAlmText:='Transfer Out Time Out While Conveyor Exit With Clamper',sRcyText:='Timeout Expired Before Operation Completed. Transmission Abnormal. Remove the Obstacle (If Exists) To Resume Operation.'),(sAlmText:='Transfer Out Time Out While Exiting Magazine',sRcyText:='Timeout Expired Before Operation Completed. Transmission Abnormal. Remove the Obstacle (If Exists) To Resume Operation.'),(sAlmText:='Transfer Out Time Out While Conveyor Exit With Clamper',sRcyText:='Timeout Expired Before Operation Completed. Transmission Abnormal. Remove the Obstacle (If Exists) To Resume Operation.'),(sAlmText:='Clamper Clamp Sensor On Time Out In Clamp Check While Conveyor Enter With Clamper',sRcyText:='Sensor Timeout Expired Before Operation Completed. Sensor Operation Is Abnormal. Solve The Error To Resume Operation.'),(sAlmText:='Clamper Unclamp Sensor Off Time Out In Clamp Check While Conveyor Enter With Clamper',sRcyText:='Sensor Timeout Expired Before Operation Completed. Sensor Operation Is Abnormal. Solve The Error To Resume Operation.'),(sAlmText:='Clamper Clamp Safety Sensor Error In Clamp Check While Conveyor Enter With Clamper',sRcyText:='Safety System Has Been Triggered. All Operations Are Disable. Remove the Obstacle That Triggered The Safety Interlock To Resume Operation.'),(sAlmText:='Transfer In Time Out While Entering Magazine',sRcyText:='Timeout Expired Before Operation Completed. Transmission Abnormal. Remove the Obstacle (If Exists) To Resume Operation.'),(sAlmText:='Clamper Clamp Sensor Off Time Out In Unclamp Check While Conveyor Initial With Clamper',sRcyText:='Sensor Timeout Expired Before Operation Completed. Sensor Operation Is Abnormal. Solve The Error To Resume Operation.'),(sAlmText:='Clamper Unclamp Sensor On Time Out In Unclamp Check While Conveyor Initial With Clamper',sRcyText:='Sensor Timeout Expired Before Operation Completed. Sensor Operation Is Abnormal. Solve The Error To Resume Operation.'),(sAlmText:='Clamper Unclamp Safety Sensor Error In Unclamp Check While Conveyor Initial With Clamper',sRcyText:='Safety System Has Been Triggered. All Operations Are Disable. Remove the Obstacle That Triggered The Safety Interlock To Resume Operation.'),(sAlmText:='Magazine Detected But Not Present At Outlet Sensor (L - R) While Conveyor Initial With Clamper',sRcyText:='Operation Interrupted By Undetected Magazine. Adjusting The Magazine Or Remove The Present Magazine To Resume Operation.'),(sAlmText:='Magazine Detected But Not Present At Outlet Sensor (R - L) While Conveyor Initial With Clamper',sRcyText:='Operation Interrupted By Undetected Magazine. Adjusting The Magazine Or Remove The Present Magazine To Resume Operation.'),(sAlmText:='Clamper Clamp Sensor On Time Out In Clamp Check While Conveyor Initial With Clamper',sRcyText:='Sensor Timeout Expired Before Operation Completed. Sensor Operation Is Abnormal. Solve The Error To Resume Operation.'),(sAlmText:='Clamper Unclamp Sensor Off Time Out In Clamp Check While Conveyor Initial With Clamper',sRcyText:='Sensor Timeout Expired Before Operation Completed. Sensor Operation Is Abnormal. Solve The Error To Resume Operation.'),(sAlmText:='Clamper Clamp Safety Sensor Error In Clamp Check While Conveyor Initial With Clamper',sRcyText:='Safety System Has Been Triggered. All Operations Are Disable. Remove the Obstacle That Triggered The Safety Interlock To Resume Operation.'),(sAlmText:='Magazine Not Detected While Pre-Exiting Magazine',sRcyText:='Operation Interrupted By Undetected Magazine. Adjusting The Magazine Or Remove The Present Magazine To Resume Operation.'),53((0))];
END_VAR
(**)
(*Local Output*)
VAR
	bHvMag : BOOL := FALSE;
	bMtrSigOnOrLToR : BOOL := FALSE;
	bMtrDirOrRToL : BOOL := FALSE;
	bClprClampCtrl : BOOL;
	bClprTwoOutputControl : BOOL := FALSE;
END_VAR
(**)
(*Local Input*)
VAR
	udiRstErr : UDINT := 0;
	bPrep : BOOL := TRUE;
	bEn : BOOL := TRUE;
	bDis : BOOL := FALSE;
	bManual : BOOL := FALSE;
	bOnDirMod : BOOL := FALSE;
	diInitTm : DINT := 10000;
	tMtrOffDlyTm : TIME := T#0S;
	diTxInTimeOut : DINT := 10000;
	diTxOutTimeOut : DINT := 10000;
	eDirection : eConvDir := ConvDirLToR;
	bLeftSen : BOOL := FALSE;
	bRightSen : BOOL := FALSE;
	bClprClampSen : BOOL := FALSE;
	bClprUnclampSen : BOOL := FALSE;
	bClprClampSafetySen : BOOL := TRUE;
	bClprUnclampSafetySen : BOOL := TRUE;
	sProgNm : STRING[15] := 'MagConv';
	tClprClampTO : TIME := T#20s;
	tClprUnclampTO : TIME := T#20s;
	fbSenOn1 : TON := (PT:=T#1.5s);
	bNtSettingsLoadDone : BOOL := TRUE;
END_VAR
(**)
(*Local*)
VAR
	bRstErr : BOOL;
	udiRstErrOld : UDINT;
	bInitDone : BOOL;
	bInitialDone : BOOL;
	bReachEnd : BOOL;
	usiStep : USINT;
	eStatOld : eMagConvAction := MagConvActIdle;
	fbInit : fbConvSenToSenTm;
	fbEnt : fbConvSenToSen;
	fbPreExit : fbConvSenToSenTm;
	fbExit : fbConvSenToSenOff;
	fbExit1 : fbConvSenToSenOff1;
	fbStop : fbConvMtrOff;
	fbClprClampChk : fbPneuExtRetSenExtChk;
	fbClprUnclampChk : fbPneuExtRetSenRetChk;
	fbClprDlyTm : TON;
	udiModuleNum : UDINT := 1801;
END_VAR
```

#### Act_InitGlobal.st
```iecst
(** 2019-04-09 **)
ACTION Act_InitGlobal:

	(* Always Change If Project Change *)

	//Pass Data To Link
	p_bLinkOpsRun ACCESS p_OpsRun;

	p_bLinkDISafetyRlySig ACCESS p_DISafetyRlySig;
	p_diLinkLifterActualPos ACCESS p_LifterBtmActualPos;
	p_diLinkLifterBtmPos ACCESS p_McParamLifterBtmPos;
	p_diLinkLifterTopPos ACCESS p_McParamLifterTopPos;
//	p_bLinkOpsInitULDStepInitDone ACCESS p_OpsInitULDStepInitDone;
	p_bLinkOpsLifMagULStepExtMag1 ACCESS p_OpsLifMagULStepExtMag1;

	//Pass Data To Internal Use
	p_bPrep ACCESS p_NtParamProjLifter2Prep;
	p_udiRstErr ACCESS p_RstErrReset;
	p_bManual ACCESS p_UIMnlMod;
	p_bOnDirMod ACCESS p_NtParamLifterMagOnDirMod;
	p_diInitTm ACCESS p_McParamLifterMagConvRunTmOut;
	p_diTxInTimeOut ACCESS p_McParamLifterMagConvRunTmOut;
	p_diTxOutTimeOut ACCESS p_McParamLifterMagConvRunTmOut;
	p_eDirection ACCESS p_NtParamProjLifterMagConvDir;
	p_tMtrOffDlyTm ACCESS p_NtParamLifterMagMtrOffDlyTm;
	p_bClprClampSen ACCESS p_DIMag1FixedClampRS;
	p_bClprUnclampSen ACCESS p_DIMag1FixedUnclampRS;
	p_sProgNm ACCESS p_NtParamLifterMagProgNm;
	p_bNtSettingsLoadDone ACCESS p_StartupNtSettingsLoadDone;

	// chuanyee Add
	p_bMagPresentSen ACCESS p_DILifterLmtSW;
	(* Always Change If Project Change *)

END_ACTION
```

#### Act_Link.st
```iecst
(** 2019-03-29 **)
ACTION Act_Link:

	IF (p_eAct = MagConvActEntClpStop OR p_eAct = MagConvActEnt OR p_eAct = MagConvActExitClpr OR p_eAct = MagConvActExit) AND (ABS(p_diLinkLifterActualPos - p_diLinkLifterTopPos))<500 THEN
		p_bLeftSen ACCESS p_DILifterLmtSW;
		p_bRightSen ACCESS p_DIInMagConvExtSen;
	ELSIF (p_eAct = MagConvActExitClpr OR p_eAct = MagConvActExit) OR p_bLinkOpsLifMagULStepExtMag1 THEN //(ABS(p_diLinkLifterActualPos - p_diLinkLifterBtmPos))<500 THEN
		p_bLeftSen ACCESS p_DILifterLmtSW;
		p_bRightSen ACCESS p_DIOutMagConvEntSen;

	ELSIF (p_eAct = MagConvActInitClpStop) AND eStatus <> Done THEN

		fbLeftSenOn(IN := TRUE, PT := T#5s);
		IF p_bMagPresentSen AND fbLeftSenOn.Q = FALSE AND p_bLeftSen THEN
			p_bLeftSen	:= FALSE;
		END_IF
		IF p_bMagPresentSen AND fbLeftSenOn.Q THEN
			p_bLeftSen  := TRUE;
		END_IF

		p_bRightSen ACCESS ADR(bRightSen);

	ELSIF (p_eAct = MagConvActInitClpStop) AND eStatus = Done THEN
		p_bLeftSen		:= FALSE;
		fbLeftSenOn(IN := FALSE);
		p_bRightSen ACCESS ADR(bRightSen);

	ELSE
		IF p_bMagPresentSen THEN
			fbLeftSenOnChk(IN := p_bMagPresentSen, PT := T#3s);
			IF fbLeftSenOnChk.Q THEN
				p_bLeftSen := p_bMagPresentSen;
				fbLeftSenOnChk(IN := FALSE);
			ELSE
			END_IF
			p_bRightSen ACCESS ADR(bRightSen);
		ELSE

			p_bLeftSen := p_bMagPresentSen;
			p_bRightSen ACCESS ADR(bRightSen);
		END_IF
	END_IF

	fbClprDlyTm.PT		:= p_tMtrOffDlyTm / 2;

	IF p_bLinkDISafetyRlySig = FALSE THEN
		bClprClampCtrl := FALSE;
		fbLeftSenOnChk(IN := FALSE);
		fbLeftSenOn(IN := FALSE);
	END_IF

	IF EDGEPOS(eStatus = Error) THEN
		bMtrSigOnOrLToR	:= FALSE;
		bMtrDirOrRToL	:= FALSE;
		fbLeftSenOnChk(IN := FALSE);
		fbLeftSenOn(IN := FALSE);
	END_IF

END_ACTION
```

#### Act_LinkAction.st
```iecst
(** 2019-04-09 **)
ACTION Act_LinkAction:

	IF p_bLinkOpsRun = TRUE AND p_OpsLifMagULLifterConvAct <> 0 THEN
//		IF p_bLinkOpsInitULDStepInitDone = FALSE THEN
//			p_eAct ACCESS p_OpsInitULDLifterMagConvAct;
//		ELSE
			p_eAct ACCESS p_OpsLifMagULLifterConvAct;
//		END_IF
	ELSIF p_bManual = TRUE THEN
		p_eAct ACCESS p_UILifterMagConvAct;
	ELSE
		p_eAct ACCESS ADR(eAct);
	END_IF

END_ACTION
```

#### Cyclic.st
```iecst
(** 2019-03-29 **)
PROGRAM _CYCLIC

	IF bInitDone = FALSE THEN
		bInitDone	:= TRUE;

		Act_InitLocal;
		Act_InitGlobal;

	ELSIF bInitialDone = FALSE THEN
		IF p_bNtSettingsLoadDone = TRUE THEN
			bInitialDone	:= TRUE;

			Act_Initial;
		END_IF

	ELSE

		Act_RstErr;
		Act_LinkAction;
		Act_Action;
		Act_LinkEn;

		IF (p_bPrep = TRUE) AND (p_bEn = TRUE) AND (p_bDis = FALSE) THEN
			Act_Link;
			Act_Main;
		ELSE
			IF eStat <> MagConvActIdle THEN
				eStatus	:= Done;
			ELSE
				eStatus	:= Idle;
			END_IF
		END_IF

		Act_Alarm;

	END_IF

END_PROGRAM
```

#### Init.st
```iecst
(** 2019-03-25 **)
PROGRAM _INIT

	(* Always Change If Project Change *)

	//Physical Configuration
//	tMtrOffDlyTm	:= T#0s;

	//Pass Address To Global Address For External Use
	//Action, State & Status
	p_LifterMagConvStat			:= ADR(eStat);
	p_LifterMagConvStatus		:= ADR(eStatus);
	p_LifterMagConvStatTxt		:= ADR(sStatTxt);

	//Alarm
	p_LifterMagConvAlmData		:= ADR(tyAlmData);

	//Output
	p_LifterMagConvHvMag				:= ADR(bHvMag);
	p_LifterMagConvMtrSigOnOrLToR		:= ADR(bMtrSigOnOrLToR);
	p_LifterMagConvMtrDirOrRToL			:= ADR(bMtrDirOrRToL);

	p_LifterMagConvClprClampCtrl		:= ADR(bClprClampCtrl);
	p_LifterMagConvClprTwoOutputCtrl	:= ADR(bClprTwoOutputControl);

	(* Always Change If Project Change *)

END_PROGRAM
```

### InMagConv2.var - Change By Project
```iecst
(*2019-03-25*)
(**)
(*Action & State & Status*)
VAR
	p_InMagConv2Stat : UDINT;
	p_InMagConv2Status : UDINT;
	p_InMagConv2StatTxt : UDINT;
END_VAR
(**)
(*Alarm*)
VAR
	p_InMagConv2AlmData : UDINT;
END_VAR
(**)
(*Output*)
VAR
	p_InMagConv2HvMag : UDINT;
	p_InMagConv2MtrSigOnOrLToR : UDINT;
	p_InMagConv2MtrDirOrRToL : UDINT;
	p_InMagConv2ClprClampCtrl : UDINT;
	p_InMagConv2ClprTwoOutputControl : UDINT;
END_VAR
```

### Program Logical/MagConv_TopBtm/InMagConv2 (IEC) - 1.00.0 - NtConv v5.00.0 , NtPneu v5.00.0

#### InputRef.var
```iecst
(*2019-03-25*)
(**)
(*General*)
VAR
	p_eAct : REFERENCE TO eMagConvAction;
	p_udiRstErr : REFERENCE TO UDINT;
	p_bPrep : REFERENCE TO BOOL;
	p_bEn : REFERENCE TO BOOL;
	p_bDis : REFERENCE TO BOOL;
END_VAR
(**)
(*Configuration*)
VAR
	p_bManual : REFERENCE TO BOOL;
	p_bOnDirMod : REFERENCE TO BOOL;
	p_diInitTm : REFERENCE TO DINT;
	p_tMtrOffDlyTm : REFERENCE TO TIME;
	p_diTxInTimeOut : REFERENCE TO DINT;
	p_diTxOutTimeOut : REFERENCE TO DINT;
	p_eDirection : REFERENCE TO eConvDir;
	p_sProgNm : REFERENCE TO STRING[15];
	p_tClprClampTO : REFERENCE TO TIME;
	p_tClprUnclampTO : REFERENCE TO TIME;
	p_bNtSettingsLoadDone : REFERENCE TO BOOL;
END_VAR
(**)
(*Input*)
VAR
	p_bLeftSen : REFERENCE TO BOOL;
	p_bRightSen : REFERENCE TO BOOL;
	p_bClprClampSen : REFERENCE TO BOOL;
	p_bClprUnclampSen : REFERENCE TO BOOL;
	p_bClprClampSafetySen : REFERENCE TO BOOL;
	p_bClprUnclampSafetySen : REFERENCE TO BOOL;
END_VAR
```

#### InputRef_Link.var
```iecst
(*2019-04-09*)
(**)
VAR
	p_bLinkOpsRun : REFERENCE TO BOOL;
END_VAR
(**)
VAR
	p_bLinkDISafetyRlySig : REFERENCE TO BOOL;
	p_bLinkOpsInitULDStepInitDone2 : REFERENCE TO BOOL;
	p_bLinkInMagConv2MidSen : REFERENCE TO BOOL;
	p_bLinkInMagConv2ExtSen : REFERENCE TO BOOL;
	p_bLinkLifter2LmtSW : REFERENCE TO BOOL;
	fbLeftSenOnChk : TON;
	p_bLinkOpsInMagConv2StepEntToMid : REFERENCE TO BOOL;
END_VAR
```

#### Act_Action.st
```iecst
(** 2019-03-25 **)
ACTION Act_Action:

	//Reset Error
	IF (eStatus = Error) AND bRstErr THEN
		p_eAct	:= MagConvActIdle;
		eStat	:= MagConvActIdle;
	END_IF

	//Set p_eAct
	IF eStatus = Idle OR eStatus = Busy OR eStatus = Done THEN
		eStat	:= p_eAct;
	END_IF

END_ACTION
```

#### Act_InitGlobal.st
```iecst
(** 2019-04-09 **)
ACTION Act_InitGlobal:

	(* Always Change If Project Change *)

	//Pass Data To Links
	p_bLinkOpsRun ACCESS p_OpsRun;

	p_bLinkDISafetyRlySig ACCESS p_DISafetyRlySig;
	p_bLinkOpsInitULDStepInitDone2 ACCESS p_OpsLifMagULStepInitDone2;
	p_bLinkInMagConv2MidSen ACCESS p_DIInMagConv2MidSen;
	p_bLinkInMagConv2ExtSen ACCESS p_DIInMagConv2ExtSen;
	p_bLinkLifter2LmtSW ACCESS p_DILifter2LmtSW;
	p_bLinkOpsInMagConv2StepEntToMid ACCESS p_OpsInMagConv2StepEntToMid;

	//Pass Data To Internal Use
	p_udiRstErr ACCESS p_RstErrReset;
	p_bManual ACCESS p_UIMnlMod;
	p_bOnDirMod ACCESS p_NtParamInMagConv2OnDirMod;
	p_tMtrOffDlyTm ACCESS p_NtParamInMagConv2MtrOffDlyTm;
	p_diInitTm ACCESS p_McParamInMagConv2RunTmOut;
	p_diTxInTimeOut ACCESS p_McParamInMagConv2RunTmOut;
	p_diTxOutTimeOut ACCESS p_McParamInMagConv2RunTmOut;
//	p_bRightSen ACCESS p_DIInMagConv2MidSen;
	p_eDirection ACCESS p_NtParamProjInMagConv2Dir;
	p_sProgNm ACCESS p_NtParamInMagConv2ProgNm;
	p_bNtSettingsLoadDone ACCESS p_StartupNtSettingsLoadDone;

	(* Always Change If Project Change *)

END_ACTION
```

#### Act_Link.st
```iecst
(** 2019-03-29 **)
ACTION Act_Link:
	//InMag unloader -> R-L
	IF p_eAct = MagConvActInit OR p_eAct = MagConvActEnt THEN
		IF p_bLinkOpsInMagConv2StepEntToMid THEN
			p_bRightSen ACCESS p_DIInMagConv2EntSen;
			p_bLeftSen		:= p_bLinkInMagConv2MidSen;
		ELSE
			p_bRightSen ACCESS p_DIInMagConv2MidSen;
			p_bLeftSen		:= p_bLinkInMagConv2ExtSen;
		END_IF

	//	p_bRightSen ACCESS p_DIInMagConvMidSen;
	ELSIF p_eAct = MagConvActExit THEN
		p_bLeftSen		:= p_bLinkLifter2LmtSW = FALSE;
		p_bRightSen ACCESS p_DIInMagConv2MidSen;
	ELSE
		p_bRightSen ACCESS p_DIInMagConv2MidSen;
	END_IF

	IF EDGEPOS(eStatus = Error) THEN
		bMtrSigOnOrLToR	:= FALSE;
		bMtrDirOrRToL	:= FALSE;
	END_IF

END_ACTION
```

#### Act_LinkAction.st
```iecst
(** 2019-04-09 **)
ACTION Act_LinkAction:

	IF p_bLinkOpsRun = TRUE AND p_OpsInMagConv2Act <> 0 THEN
//		IF p_bLinkOpsInitULDStepInitDone2 = FALSE THEN
//			p_eAct ACCESS p_OpsLifMagULInMagConv2Act;
//		ELSE
			p_eAct ACCESS p_OpsInMagConv2Act;
//		END_IF
	ELSIF p_bManual = TRUE THEN
		p_eAct ACCESS p_UIInMagConv2Act;
	ELSE
		p_eAct ACCESS ADR(eAct);
	END_IF

END_ACTION
```

#### Init.st
```iecst
(** 2019-03-25 **)
PROGRAM _INIT

	(* Always Change If Project Change *)

	//Pass Address To Global Address For External Use
	//Action, State & Status
	p_InMagConv2Stat		:= ADR(eStat);
	p_InMagConv2Status	:= ADR(eStatus);
	p_InMagConv2StatTxt	:= ADR(sStatTxt);

	//Alarm
	p_InMagConv2AlmData	:= ADR(tyAlmData);

	//Output
	p_InMagConv2HvMag				:= ADR(bHvMag);
	p_InMagConv2MtrSigOnOrLToR		:= ADR(bMtrSigOnOrLToR);
	p_InMagConv2MtrDirOrRToL		:= ADR(bMtrDirOrRToL);

	p_InMagConv2ClprClampCtrl		:= ADR(bClprClampCtrl);
	p_InMagConv2ClprTwoOutputControl:= ADR(bClprTwoOutputControl);

	(* Always Change If Project Change *)

END_PROGRAM
```

### OutMagConv2.var - Change By Project
```iecst
(*2019-03-25*)
(**)
(*Action & State & Status*)
VAR
	p_OutMagConv2Stat : UDINT;
	p_OutMagConv2Status : UDINT;
	p_OutMagConv2StatTxt : UDINT;
END_VAR
(**)
(*Alarm*)
VAR
	p_OutMagConv2AlmData : UDINT;
END_VAR
(**)
(*Output*)
VAR
	p_OutMagConv2HvMag : UDINT;
	p_OutMagConv2MtrSigOnOrLToR : UDINT;
	p_OutMagConv2MtrDirOrRToL : UDINT;
	p_OutMagConv2ClprClampCtrl : UDINT;
	p_OutMagConv2ClprTwoOutControl : UDINT;
END_VAR
```

### Program Logical/MagConv_TopBtm/OutMagConv2 (IEC) - 1.00.0 - NtConv v5.00.0 , NtPneu v5.00.0

#### InputRef_Link.var
```iecst
(*2019-04-09*)
(**)
VAR
	p_bLinkOpsRun : REFERENCE TO BOOL;
END_VAR
(**)
VAR
	p_bLinkDISafetyRlySig : REFERENCE TO BOOL;
	fbOutMagConvStopTm : TON;
	bTmr : BOOL;
	p_tyLinkDI : REFERENCE TO tyDigitalInputSettings;
	p_bLinkOpsInitULDStepInitDone2 : REFERENCE TO BOOL;
	p_bLinkOpsOutMagConStepEntMag : REFERENCE TO BOOL;
	p_bLinkOpsOutMagConStepEntMidMag : REFERENCE TO BOOL;
END_VAR
```

#### Act_InitGlobal.st
```iecst
(** 2019-04-09 **)
ACTION Act_InitGlobal:

	(* Always Change If Project Change *)

	//Pass Data To Link
	p_bLinkOpsRun ACCESS p_OpsRun;

	p_bLinkDISafetyRlySig ACCESS p_DISafetyRlySig;
	p_tyLinkDI ACCESS p_NtParamDISettings;
	p_bLinkOpsInitULDStepInitDone2 ACCESS p_OpsLifMagULStepInitDone2;
	p_bLinkOpsOutMagConStepEntMag ACCESS p_OpsOutMagConv2StepEntMag;
	p_bLinkOpsOutMagConStepEntMidMag ACCESS p_OpsOutMagConv2StepEntMidMag;

	//Pass Data To Internal Use
	p_udiRstErr ACCESS p_RstErrReset;
	p_bManual ACCESS p_UIMnlMod;
	p_bOnDirMod ACCESS p_NtParamOutMagConv2OnDirMod;
	p_tMtrOffDlyTm ACCESS p_NtParamOutMagConv2MtrOffDlyTm;
	p_diInitTm ACCESS p_McParamOutMagConv2RunTmOut;
	p_diTxInTimeOut ACCESS p_McParamOutMagConv2RunTmOut;
	p_diTxOutTimeOut ACCESS p_McParamOutMagConv2RunTmOut;
	p_eDirection ACCESS p_NtParamProjOutMagConv2Dir;
	p_bLeftSen ACCESS p_DIOutMagConv2EntSen;
	p_sProgNm ACCESS p_NtParamOutMagConv2ProgNm;
	p_bNtSettingsLoadDone ACCESS p_StartupNtSettingsLoadDone;

	(* Always Change If Project Change *)

END_ACTION
```

#### Act_Link.st
```iecst
(** 2019-03-29 **)
ACTION Act_Link:

	IF p_tyLinkDI.diOutMagConvExtSen = 0 THEN
		IF EDGENEG (p_bLeftSen) AND (eStat = MagConvActEnt) THEN
			bTmr := TRUE;
		END_IF

		IF bTmr	= TRUE THEN
			fbOutMagConvStopTm(IN := TRUE, PT:=T#3500ms);

			IF fbOutMagConvStopTm.Q THEN
				fbOutMagConvStopTm(IN:=FALSE);

				p_bRightSen := TRUE;
				bTmr		:= FALSE;
			END_IF
		END_IF

		IF (eStat = MagConvActEnt AND eStatus = Done) THEN
			p_bRightSen		:= FALSE;
		END_IF

	ELSIF p_bLinkOpsOutMagConStepEntMag THEN 	//add
		p_bRightSen ACCESS p_DIOutMagConv2ExtSen;
	ELSIF p_bLinkOpsOutMagConStepEntMidMag THEN //add
		p_bRightSen ACCESS p_DIOutMagConv2MidSen;
	ELSE
		p_bRightSen ACCESS p_DIOutMagConv2ExtSen;
	END_IF

	IF EDGEPOS(eStatus = Error) THEN
		bMtrSigOnOrLToR	:= FALSE;
		bMtrDirOrRToL	:= FALSE;
	END_IF

END_ACTION
```

#### Act_LinkAction.st
```iecst
(** 2019-04-09 **)
ACTION Act_LinkAction:

	IF p_bLinkOpsRun = TRUE AND p_OpsOutMagConv2Act <> 0 THEN
//		IF p_bLinkOpsInitULDStepInitDone2 = FALSE THEN
//			p_eAct ACCESS p_OpsLifMagULOutMagConv2Act;
//		ELSE
			p_eAct ACCESS p_OpsOutMagConv2Act;
//		END_IF
	ELSIF p_bManual = TRUE THEN
		p_eAct ACCESS p_UIOutMagConv2Act;
	ELSE
		p_eAct ACCESS ADR(eAct);
	END_IF

END_ACTION
```

#### Init.st
```iecst
(** 2019-03-25 **)
PROGRAM _INIT

	(* Always Change If Project Change *)

	//Pass Address To Global Address For External Use
	//Action, State & Status
	p_OutMagConv2Stat		:= ADR(eStat);
	p_OutMagConv2Status		:= ADR(eStatus);
	p_OutMagConv2StatTxt		:= ADR(sStatTxt);

	//Alarm
	p_OutMagConv2AlmData		:= ADR(tyAlmData);

	//Output
	p_OutMagConv2HvMag					:= ADR(bHvMag);
	p_OutMagConv2MtrSigOnOrLToR			:= ADR(bMtrSigOnOrLToR);
	p_OutMagConv2MtrDirOrRToL			:= ADR(bMtrDirOrRToL);

	p_OutMagConv2ClprClampCtrl			:= ADR(bClprClampCtrl);
	p_OutMagConv2ClprTwoOutControl	:= ADR(bClprTwoOutputControl);

	(* Always Change If Project Change *)

END_PROGRAM
```

### LifterMagConv2.var - Change By Project
```iecst
(*2019-03-25*)
(**)
(*Action & State & Status*)
VAR
	p_LifterMagConv2Stat : UDINT;
	p_LifterMagConv2Status : UDINT;
	p_LifterMagConv2StatTxt : UDINT;
END_VAR
(**)
(*Alarm*)
VAR
	p_LifterMagConv2AlmData : UDINT;
END_VAR
(**)
(*Output*)
VAR
	p_LifterMagConv2HvMag : UDINT;
	p_LifterMagConv2MtrSigOnOrLToR : UDINT;
	p_LifterMagConv2MtrDirOrRToL : UDINT;
	p_LifterMagConv2ClprClampCtrl : UDINT;
	p_LifterMagConv2ClprTwoOutCtrl : UDINT;
END_VAR
```

### Program Logical/MagConv_TopBtm/LifterMagConv2 (IEC) - 1.00.0 - NtConv v5.00.0 , NtPneu v5.00.0

#### InputRef_Link.var
```iecst
(*2019-04-09*)
(**)
(*External*)
VAR
	p_bLinkOpsRun : REFERENCE TO BOOL;
END_VAR
(**)
VAR
	p_bLinkDISafetyRlySig : REFERENCE TO BOOL;
	p_diLinkLifterActualPos : REFERENCE TO DINT;
	p_diLinkLifterBtmPos : REFERENCE TO DINT;
	p_diLinkLifterTopPos : REFERENCE TO DINT;
	p_bLinkOpsInitULDStepInitDone : REFERENCE TO BOOL;
	p_bLinkTopMagConvEntSen : REFERENCE TO BOOL;
	p_bLinkOpsLifMagULStepExtMag2 : REFERENCE TO BOOL;
END_VAR
(**)
VAR
	fbLeftSenOnChk : TON;
	fbLeftSenOn : TON;
END_VAR
```

#### Act_Alarm.st
```iecst
(** 2019-03-25 **)
ACTION Act_Alarm:

	//Error
	IF EDGEPOS(eStatus = Error) THEN

		tyAlmData.sProgNm		:= p_sProgNm;
		tyAlmData.udiCode		:= udiStatus;
		tyAlmData.eSeverity		:= AlmSeverityError;
		tyAlmData.udiRunTime	:= tyAlmData.udiRunTime + 1;
		tyAlmData.bAlm			:= TRUE;
		tyAlmData.udiModuleNum  := udiModuleNum;
		g_sMagConvProgNm		:= p_sProgNm;

		//Get Error Message
		IF tyAlmData.udiCode < 10000 OR tyAlmData.udiCode > 10099 THEN
			tyAlmData.sAlmMsg	:= 'Unknown';
			tyAlmData.sRcyMsg	:= 'Unknown';
		ELSE
			tyAlmData.sAlmMsg	:= a_tyAlmText[tyAlmData.udiCode].sAlmText;
			tyAlmData.sRcyMsg	:= a_tyAlmText[tyAlmData.udiCode].sRcyText;
		END_IF

		sStatTxt	:= tyAlmData.sAlmMsg;

	ELSIF bRstErr AND (tyAlmData.udiCode <> 0) THEN

		tyAlmData.udiCode	:= 0;
		tyAlmData.eSeverity	:= AlmSeverityNA;
		tyAlmData.sAlmMsg	:= '';
		tyAlmData.sRcyMsg	:= '';
		tyAlmData.bAlm			:= FALSE;
		sStatTxt	:= a_sStatText[eStat];

	END_IF

END_ACTION
```

#### Act_InitGlobal.st
```iecst
(** 2019-04-09 **)
ACTION Act_InitGlobal:

	(* Always Change If Project Change *)

	//Pass Data To Link
	p_bLinkOpsRun ACCESS p_OpsRun;

	p_bLinkDISafetyRlySig ACCESS p_DISafetyRlySig;
	p_diLinkLifterActualPos ACCESS p_Lifter2ActualPos;
	p_diLinkLifterBtmPos ACCESS p_McParamLifterBtmPos2;
	p_diLinkLifterTopPos ACCESS p_McParamLifterTopPos2;
//	p_bLinkOpsInitULDStepInitDone ACCESS p_OpsInitULDStepInitDone;
	p_bLinkOpsLifMagULStepExtMag2 ACCESS p_OpsLifMagULStepExtMag2;

	//Pass Data To Internal Use
	p_bPrep ACCESS p_NtParamProjLifter2Prep;
	p_udiRstErr ACCESS p_RstErrReset;
	p_bManual ACCESS p_UIMnlMod;
	p_bOnDirMod ACCESS p_NtParamLifterMag2OnDirMod;
	p_diInitTm ACCESS p_McParamLifterMagConv2RunTmOut;
	p_diTxInTimeOut ACCESS p_McParamLifterMagConv2RunTmOut;
	p_diTxOutTimeOut ACCESS p_McParamLifterMagConv2RunTmOut;
	p_eDirection ACCESS p_NtParamProjLifterMagConv2Dir;
	p_tMtrOffDlyTm ACCESS p_NtParamLifterMag2MtrOffDlyTm;
	p_bClprClampSen ACCESS p_DIMag2FixedClampRS; //Clamp
	p_bClprUnclampSen ACCESS p_DIMag2FixedUnclampRS;
	p_sProgNm ACCESS p_NtParamLifterMag2ProgNm;
	p_bNtSettingsLoadDone ACCESS p_StartupNtSettingsLoadDone;

	// chuanyee Add
	p_bMagPresentSen ACCESS p_DILifter2LmtSW;
	(* Always Change If Project Change *)

END_ACTION
```

#### Act_Initial.st
```iecst
(** 2019-05-28 **)
ACTION Act_Initial:

	//Initial
	sStatTxt	:= a_sStatText[eStat];

	fbInit.bOnDirMod	:= p_bOnDirMod;
	fbInit.bStartSen	:= TRUE;
	fbInit.tMtrOffDlyTm	:= p_tMtrOffDlyTm;
	fbInit(bEn := FALSE);

	fbEnt.bOnDirMod		:= p_bOnDirMod;
	fbEnt.bStartSen		:= TRUE;
	fbEnt.tMtrOffDlyTm	:= p_tMtrOffDlyTm;
	fbEnt(bEn := FALSE);

	fbPreExit.bOnDirMod		:= p_bOnDirMod;
	fbPreExit.bStartSen		:= TRUE;
	fbPreExit.tMtrOffDlyTm	:= p_tMtrOffDlyTm;
	fbPreExit(bEn := FALSE);

	fbExit.bOnDirMod	:= p_bOnDirMod;
	fbExit.bStartSen	:= TRUE;
	fbExit.tMtrOffDlyTm	:= p_tMtrOffDlyTm;
	fbExit(bEn := FALSE);

	fbExit1.bOnDirMod		:= p_bOnDirMod;
	fbExit1.bStartSen		:= TRUE;
	fbExit1.tMtrOffDlyTm	:= p_tMtrOffDlyTm;
	fbExit1(bEn := FALSE);

	fbStop(bEn := FALSE);

	fbClprClampChk.tTimeOut	:= p_tClprClampTO;
	fbClprClampChk(bEn := FALSE);

	fbClprUnclampChk.tTimeOut	:= p_tClprUnclampTO;
	fbClprUnclampChk(bEn := FALSE);

	fbClprDlyTm.PT	:= p_tMtrOffDlyTm / 2;
	fbClprDlyTm(IN := FALSE);

END_ACTION
```

#### Act_Link.st
```iecst
(** 2019-03-29 **)
ACTION Act_Link:

	IF (p_eAct = MagConvActEntClpStop OR p_eAct = MagConvActEnt OR p_eAct = MagConvActExitClpr OR p_eAct = MagConvActExit) AND (ABS(p_diLinkLifterActualPos - p_diLinkLifterTopPos))<500 THEN
		p_bLeftSen ACCESS p_DILifter2LmtSW;
		p_bRightSen ACCESS p_DIInMagConv2ExtSen;
	ELSIF (p_eAct = MagConvActExitClpr OR p_eAct = MagConvActExit) OR p_bLinkOpsLifMagULStepExtMag2 THEN //AND (ABS(p_diLinkLifterActualPos - p_diLinkLifterBtmPos))<500 THEN
		p_bLeftSen ACCESS p_DILifter2LmtSW;
		p_bRightSen ACCESS p_DIOutMagConv2EntSen;

	ELSIF (p_eAct = MagConvActInitClpStop) AND eStatus <> Done THEN

		fbLeftSenOn(IN := TRUE, PT := T#5s);
		IF p_bMagPresentSen AND fbLeftSenOn.Q = FALSE AND p_bLeftSen THEN
			p_bLeftSen	:= FALSE;
		END_IF
		IF p_bMagPresentSen AND fbLeftSenOn.Q THEN
			p_bLeftSen  := TRUE;
		END_IF

		p_bRightSen ACCESS ADR(bRightSen);

	ELSIF (p_eAct = MagConvActInitClpStop) AND eStatus = Done THEN
		p_bLeftSen		:= FALSE;
		fbLeftSenOn(IN := FALSE);
		p_bRightSen ACCESS ADR(bRightSen);

	ELSE
		IF p_bMagPresentSen THEN
			fbLeftSenOnChk(IN := p_bMagPresentSen, PT := T#3s);
			IF fbLeftSenOnChk.Q THEN
				p_bLeftSen := p_bMagPresentSen;
				fbLeftSenOnChk(IN := FALSE);
			ELSE
			END_IF
			p_bRightSen ACCESS ADR(bRightSen);
		ELSE

			p_bLeftSen := p_bMagPresentSen;
			p_bRightSen ACCESS ADR(bRightSen);
		END_IF
	END_IF

	fbClprDlyTm.PT		:= p_tMtrOffDlyTm / 2;

	IF p_bLinkDISafetyRlySig = FALSE THEN
		bClprClampCtrl := FALSE;
		fbLeftSenOnChk(IN := FALSE);
		fbLeftSenOn(IN := FALSE);
	END_IF

	IF EDGEPOS(eStatus = Error) THEN
		bMtrSigOnOrLToR	:= FALSE;
		bMtrDirOrRToL	:= FALSE;
		fbLeftSenOnChk(IN := FALSE);
		fbLeftSenOn(IN := FALSE);
	END_IF

END_ACTION
```

#### Act_LinkAction.st
```iecst
(** 2019-04-09 **)
ACTION Act_LinkAction:

	IF p_bLinkOpsRun = TRUE THEN
//		IF p_bLinkOpsInitULDStepInitDone = FALSE THEN
//			p_eAct ACCESS p_OpsInitULDLifterMagConvAct;
//		ELSE
			p_eAct ACCESS p_OpsLifMagULLifterConv2Act;
//		END_IF
	ELSIF p_bManual = TRUE THEN
		p_eAct ACCESS p_UILifterMagConv2Act;
	ELSE
		p_eAct ACCESS ADR(eAct);
	END_IF

END_ACTION
```

#### Act_Main.st
```iecst
(** 2019-05-28 **)
ACTION Act_Main:

	IF eStatOld <> eStat THEN
		fbInit(bEn := FALSE);
		fbEnt(bEn := FALSE);
		fbPreExit(bEn := FALSE);
		fbExit(bEn := FALSE);
		fbExit1(bEn := FALSE);
		fbStop(bEn := FALSE);
		fbClprClampChk(bEn := FALSE);
		fbClprUnclampChk(bEn := FALSE);

		IF eStatOld <> MagConvActIdle
			AND eStatOld <> MagConvActSetMtrSigOnOrLToR
			AND eStatOld <> MagConvActSetMtrDirOrRToL
			AND eStatOld <> MagConvActRstMtrSigOnOrLToR
			AND eStatOld <> MagConvActRstMtrDirOrRToL
			AND eStatOld <> MagConvActSetMtrAll
			AND eStatOld <> MagConvActRstMtrAll THEN

			bMtrSigOnOrLToR	:= FALSE;
			bMtrDirOrRToL	:= FALSE;

		END_IF

		usiStep		:= 0;
		bReachEnd	:= FALSE;

		sStatTxt	:= a_sStatText[eStat];

		eStatOld	:= eStat;

		eStatus		:= Busy;
	END_IF

	//Main
	CASE eStat OF

		MagConvActIdle:
			IF EDGENEG(p_bManual) THEN
				bMtrSigOnOrLToR	:= FALSE;
				bMtrDirOrRToL	:= FALSE;
			END_IF

			eStatus	:= Idle;

		MagConvActInit:
			IF eStatus = Idle OR eStatus = Busy THEN

				eStatus	:= Busy;

				//Magazine Conveyor Init Run
				//Detect Have Magazine
				IF p_bLeftSen OR p_bRightSen THEN
					bHvMag	:= TRUE;
				ELSE
					bHvMag	:= FALSE;
				END_IF

				fbInit.bConvLToR	:= (p_eDirection = ConvDirLToR) OR (p_eDirection = ConvDirLToL);
				fbInit.tTxDlyTm		:= DINT_TO_TIME(p_diInitTm);

				IF fbInit.bConvLToR = TRUE THEN
					fbInit.bEndSen	:= p_bRightSen;
				ELSE
					fbInit.bEndSen	:= p_bLeftSen;
				END_IF

				fbInit(bEn := TRUE);

				bMtrSigOnOrLToR	:= fbInit.bMtrSigOnOrLToR;
				bMtrDirOrRToL	:= fbInit.bMtrDirOrRToL;

				IF fbInit.udiStatus = 0 THEN
					IF fbInit.bConvLToR = TRUE THEN
						IF bHvMag = TRUE AND p_bRightSen = FALSE THEN
							udiStatus	:= 10000;	//Magazine Detected But Not Present At Outlet Sensor (L - R) While Magazine Conveyor Initial
							eStatus		:= Error;
						ELSE
							eStatus	:= Done;
						END_IF
					ELSE
						IF bHvMag = TRUE AND p_bLeftSen = FALSE THEN
							udiStatus	:= 10001;	//Magazine Detected But Not Present At Outlet Sensor (R - L) While Magazine Conveyor Initial
							eStatus		:= Error;
						ELSE
							eStatus	:= Done;
						END_IF
					END_IF
				ELSIF fbInit.udiStatus < 65534 THEN
					udiStatus	:= fbInit.udiStatus;
					eStatus		:= Error;
				END_IF
			END_IF

		MagConvActInitStopClp:
			IF eStatus = Idle OR eStatus = Busy THEN

				eStatus	:= Busy;

				CASE usiStep OF
					0: //Unclamp
						bClprClampCtrl		:= FALSE;

						fbClprUnclampChk.bExtSen	:= p_bClprClampSen;
						fbClprUnclampChk.bRetSen	:= p_bClprUnclampSen;
						fbClprUnclampChk.bRetSafety	:= p_bClprUnclampSafetySen;
						fbClprUnclampChk(bEn := TRUE);

						IF fbClprUnclampChk.udiStatus = 0 THEN
							usiStep	:= 1;
						ELSIF fbClprUnclampChk.udiStatus < 65534 THEN
							bClprClampCtrl		:= TRUE;

							eStatus			:= Error;

							IF fbClprUnclampChk.udiStatus = 1504 THEN
								udiStatus	:= 10002;	//Clamper Clamp Sensor Off Time Out In Unclamp Check While Conveyor Initial With Clamper
							ELSIF fbClprUnclampChk.udiStatus = 1505 THEN
								udiStatus	:= 10003;	//Clamper Unclamp Sensor On Time Out In Unclamp Check While Conveyor Initial With Clamper
							ELSIF fbClprUnclampChk.udiStatus = 1508 THEN
								udiStatus	:= 10004;	//Clamper Unclamp Safety Sensor Error In Unclamp Check While Conveyor Initial With Clamper
							ELSE
								udiStatus	:= fbClprUnclampChk.udiStatus;
							END_IF
						END_IF

					1:	//Magazine Conveyor Init Run
						//Detect Have Magazine
						IF p_bLeftSen OR p_bRightSen THEN
							bHvMag	:= TRUE;
						ELSE
							bHvMag	:= FALSE;
						END_IF

						fbInit.bConvLToR	:= (p_eDirection = ConvDirLToR) OR (p_eDirection = ConvDirLToL);
						fbInit.tTxDlyTm		:= DINT_TO_TIME(p_diInitTm);

						IF fbInit.bConvLToR = TRUE THEN
							fbInit.bEndSen	:= p_bRightSen;
						ELSE
							fbInit.bEndSen	:= p_bLeftSen;
						END_IF

						fbInit(bEn := TRUE);

						bMtrSigOnOrLToR	:= fbInit.bMtrSigOnOrLToR;
						bMtrDirOrRToL	:= fbInit.bMtrDirOrRToL;

						IF fbInit.udiStatus = 0 THEN
							IF fbInit.bConvLToR = TRUE THEN
								IF bHvMag = TRUE AND p_bRightSen = FALSE THEN
									udiStatus	:= 10005;	//Magazine Detected But Not Present At Outlet Sensor (L - R) While Conveyor Initial With Clamper
									eStatus		:= Error;
								ELSE
									usiStep	:= 2;
								END_IF
							ELSE
								IF bHvMag = TRUE AND p_bLeftSen = FALSE THEN
									udiStatus	:= 10006;	//Magazine Detected But Not Present At Outlet Sensor (R - L) While Conveyor Initial With Clamper
									eStatus		:= Error;
								ELSE
									usiStep	:= 2;
								END_IF
							END_IF
						ELSIF fbInit.udiStatus < 65534 THEN
							udiStatus	:= fbInit.udiStatus;
							eStatus		:= Error;
						END_IF

					2:	//Check If Have Magazine

						IF bHvMag = TRUE THEN
							usiStep	:= 3;
						ELSE
							eStatus	:= Done;
						END_IF

					3:	//Clamp
						bClprClampCtrl		:= TRUE;

						fbClprClampChk.bExtSen		:= p_bClprClampSen;
						fbClprClampChk.bRetSen		:= p_bClprUnclampSen;
						fbClprClampChk.bExtSafety	:= p_bClprClampSafetySen;
						fbClprClampChk(bEn := TRUE);

						IF fbClprClampChk.udiStatus = 0 THEN
							eStatus		:= Done;
						ELSIF fbClprClampChk.udiStatus < 65534 THEN
							bClprClampCtrl		:= FALSE;

							eStatus			:= Error;

							IF fbClprClampChk.udiStatus = 1503 THEN
								udiStatus	:= 10007;	//Clamper Clamp Sensor On Time Out In Clamp Check While Conveyor Initial With Clamper
							ELSIF fbClprClampChk.udiStatus = 1506 THEN
								udiStatus	:= 10008;	//Clamper Unclamp Sensor Off Time Out In Clamp Check While Conveyor Initial With Clamper
							ELSIF fbClprClampChk.udiStatus = 1507 THEN
								udiStatus	:= 10009;	//Clamper Clamp Safety Sensor Error In Clamp Check While Conveyor Initial With Clamper
							ELSE
								udiStatus	:= fbClprClampChk.udiStatus;
							END_IF
						END_IF

				END_CASE
			END_IF

		MagConvActInitClpStop:
			IF eStatus = Idle OR eStatus = Busy THEN

				eStatus	:= Busy;

				CASE usiStep OF
					0: //Unclamp
						bClprClampCtrl		:= FALSE;

						fbClprUnclampChk.bExtSen	:= p_bClprClampSen;
						fbClprUnclampChk.bRetSen	:= p_bClprUnclampSen;
						fbClprUnclampChk.bRetSafety	:= p_bClprUnclampSafetySen;
						fbClprUnclampChk(bEn := TRUE);

						IF fbClprUnclampChk.udiStatus = 0 THEN
							usiStep	:= 1;
						ELSIF fbClprUnclampChk.udiStatus < 65534 THEN
							bClprClampCtrl		:= TRUE;

							eStatus			:= Error;

							IF fbClprUnclampChk.udiStatus = 1504 THEN
								udiStatus	:= 10038;	//Clamper Clamp Sensor Off Time Out In Unclamp Check While Conveyor Initial With Clamper
							ELSIF fbClprUnclampChk.udiStatus = 1505 THEN
								udiStatus	:= 10039;	//Clamper Unclamp Sensor On Time Out In Unclamp Check While Conveyor Initial With Clamper
							ELSIF fbClprUnclampChk.udiStatus = 1508 THEN
								udiStatus	:= 10040;	//Clamper Unclamp Safety Sensor Error In Unclamp Check While Conveyor Initial With Clamper
							ELSE
								udiStatus	:= fbClprUnclampChk.udiStatus;
							END_IF
						END_IF

					1:	//Magazine Conveyor Init Run & Clamp
						//Detect Have Magazine
						IF p_bLeftSen OR p_bRightSen THEN
							bHvMag	:= TRUE;
						ELSE
							bHvMag	:= FALSE;
						END_IF

						fbInit.bConvLToR	:= (p_eDirection = ConvDirLToR) OR (p_eDirection = ConvDirLToL);
						fbInit.tTxDlyTm		:= DINT_TO_TIME(p_diInitTm);

						IF fbInit.bConvLToR = TRUE THEN
							fbInit.bEndSen	:= p_bRightSen;
						ELSE
							fbInit.bEndSen	:= p_bLeftSen;
						END_IF

						fbInit(bEn := TRUE);

						bMtrSigOnOrLToR	:= fbInit.bMtrSigOnOrLToR;
						bMtrDirOrRToL	:= fbInit.bMtrDirOrRToL;

						IF fbInit.bEndSen = TRUE THEN
							bReachEnd	:= TRUE;
						END_IF

						IF bReachEnd = TRUE THEN
							fbClprDlyTm(IN := TRUE);

							IF fbClprDlyTm.Q = TRUE THEN
								bClprClampCtrl		:= TRUE;

								fbClprClampChk.bExtSen		:= p_bClprClampSen;
								fbClprClampChk.bRetSen		:= p_bClprUnclampSen;
								fbClprClampChk.bExtSafety	:= p_bClprClampSafetySen;
								fbClprClampChk(bEn := TRUE);
							END_IF

						END_IF

						IF (fbInit.udiStatus = 0) AND ((fbClprClampChk.udiStatus = 0) OR (bReachEnd = FALSE)) THEN
							IF fbInit.bConvLToR = TRUE THEN
								IF bHvMag = TRUE AND p_bRightSen = FALSE THEN
									udiStatus	:= 10041;	//Magazine Detected But Not Present At Outlet Sensor (L - R) While Conveyor Initial With Clamper
									eStatus		:= Error;
								ELSE
									eStatus		:= Done;
								END_IF
							ELSE
								IF bHvMag = TRUE AND p_bLeftSen = FALSE THEN
									udiStatus	:= 10042;	//Magazine Detected But Not Present At Outlet Sensor (R - L) While Conveyor Initial With Clamper
									eStatus		:= Error;
								ELSE
									eStatus		:= Done;
								END_IF
							END_IF

						ELSIF fbInit.udiStatus > 0 AND fbInit.udiStatus < 65534 THEN
							udiStatus	:= fbInit.udiStatus;
							eStatus		:= Error;

						ELSIF fbClprClampChk.udiStatus > 0 AND fbClprClampChk.udiStatus < 65534 THEN
							bClprClampCtrl		:= FALSE;

							eStatus			:= Error;

							IF fbClprClampChk.udiStatus = 1503 THEN
								udiStatus	:= 10043;	//Clamper Clamp Sensor On Time Out In Clamp Check While Conveyor Initial With Clamper
							ELSIF fbClprClampChk.udiStatus = 1506 THEN
								udiStatus	:= 10044;	//Clamper Unclamp Sensor Off Time Out In Clamp Check While Conveyor Initial With Clamper
							ELSIF fbClprClampChk.udiStatus = 1507 THEN
								udiStatus	:= 10045;	//Clamper Clamp Safety Sensor Error In Clamp Check While Conveyor Initial With Clamper
							ELSE
								udiStatus	:= fbClprClampChk.udiStatus;
							END_IF
						END_IF

				END_CASE
			END_IF

		MagConvActEnt:
			IF eStatus = Idle OR eStatus = Busy THEN

				eStatus	:= Busy;

				//Detect Have Magazine
				IF p_bLeftSen OR p_bRightSen THEN
					bHvMag	:= TRUE;
				END_IF

				//Conveyor Run
				fbEnt.bConvLToR		:= (p_eDirection = ConvDirLToR) OR (p_eDirection = ConvDirLToL);
				fbEnt.tTimeOut		:= DINT_TO_TIME(p_diTxInTimeOut);

				IF fbEnt.bConvLToR = TRUE THEN
					fbEnt.bEndSen	:= p_bRightSen;
				ELSE
					fbEnt.bEndSen	:= p_bLeftSen;
				END_IF

				fbEnt(bEn := TRUE);

				bMtrSigOnOrLToR	:= fbEnt.bMtrSigOnOrLToR;
				bMtrDirOrRToL	:= fbEnt.bMtrDirOrRToL;

				IF fbEnt.udiStatus = 0 THEN
					eStatus		:= Done;
				ELSIF fbEnt.udiStatus < 65534 THEN
					eStatus		:= Error;

					IF fbEnt.udiStatus = 1101 THEN
						udiStatus	:= 10028;	//Transfer In Time Out While Entering Magazine
					ELSE
						udiStatus	:= fbEnt.udiStatus;
					END_IF
				END_IF

			END_IF

		MagConvActEntStopClp:
			IF eStatus = Idle OR eStatus = Busy THEN

				eStatus	:= Busy;

				CASE usiStep OF
					0:
						//Detect Have Magazine
						IF p_bLeftSen OR p_bRightSen THEN
							bHvMag	:= TRUE;
						END_IF

						//Conveyor Run
						fbEnt.bConvLToR		:= (p_eDirection = ConvDirLToR) OR (p_eDirection = ConvDirLToL);
						fbEnt.tTimeOut		:= DINT_TO_TIME(p_diTxInTimeOut);

						IF fbEnt.bConvLToR = TRUE THEN
							fbEnt.bEndSen	:= p_bRightSen;
						ELSE
							fbEnt.bEndSen	:= p_bLeftSen;
						END_IF

						fbEnt(bEn := TRUE);

						bMtrSigOnOrLToR	:= fbEnt.bMtrSigOnOrLToR;
						bMtrDirOrRToL	:= fbEnt.bMtrDirOrRToL;

						IF fbEnt.udiStatus = 0 THEN
							usiStep	:= 1;
						ELSIF fbEnt.udiStatus < 65534 THEN
							eStatus		:= Error;

							IF fbEnt.udiStatus = 1101 THEN
								udiStatus	:= 10029;	//Transfer In Time Out While Entering Magazine
							ELSE
								udiStatus	:= fbEnt.udiStatus;
							END_IF
						END_IF

					1:
						bClprClampCtrl		:= TRUE;

						fbClprClampChk.bExtSen		:= p_bClprClampSen;
						fbClprClampChk.bRetSen		:= p_bClprUnclampSen;
						fbClprClampChk.bExtSafety	:= p_bClprClampSafetySen;
						fbClprClampChk(bEn := TRUE);

						IF fbClprClampChk.udiStatus = 0 THEN
							eStatus		:= Done;
						ELSIF fbClprClampChk.udiStatus < 65534 THEN
							bClprClampCtrl		:= FALSE;

							eStatus			:= Error;

							IF fbClprClampChk.udiStatus = 1503 THEN
								udiStatus	:= 10010;	//Clamper Clamp Sensor On Time Out In Clamp Check While Conveyor Enter With Clamper
							ELSIF fbClprClampChk.udiStatus = 1506 THEN
								udiStatus	:= 10011;	//Clamper Unclamp Sensor Off Time Out In Clamp Check While Conveyor Enter With Clamper
							ELSIF fbClprClampChk.udiStatus = 1507 THEN
								udiStatus	:= 10012;	//Clamper Clamp Safety Sensor Error In Clamp Check While Conveyor Enter With Clamper
							ELSE
								udiStatus	:= fbClprClampChk.udiStatus;
							END_IF
						END_IF

				END_CASE

			END_IF

		MagConvActEntClpStop:
			IF eStatus = Idle OR eStatus = Busy THEN

				eStatus	:= Busy;

				//Detect Have Magazine
				IF p_bLeftSen OR p_bRightSen THEN
					bHvMag	:= TRUE;
				END_IF

				//Conveyor Run
				fbEnt.bConvLToR		:= (p_eDirection = ConvDirLToR) OR (p_eDirection = ConvDirLToL);
				fbEnt.tTimeOut		:= DINT_TO_TIME(p_diTxInTimeOut);

				IF fbEnt.bConvLToR = TRUE THEN
					fbEnt.bEndSen	:= p_bRightSen;
				ELSE
					fbEnt.bEndSen	:= p_bLeftSen;
				END_IF

				fbEnt(bEn := TRUE);

				bMtrSigOnOrLToR	:= fbEnt.bMtrSigOnOrLToR;
				bMtrDirOrRToL	:= fbEnt.bMtrDirOrRToL;

				IF fbEnt.bEndSen = TRUE THEN
					bReachEnd	:= TRUE;
				END_IF

				IF bReachEnd = TRUE THEN
					fbClprDlyTm(IN := TRUE);

					IF fbClprDlyTm.Q = TRUE THEN
						bClprClampCtrl		:= TRUE;

						fbClprClampChk.bExtSen		:= p_bClprClampSen;
						fbClprClampChk.bRetSen		:= p_bClprUnclampSen;
						fbClprClampChk.bExtSafety	:= p_bClprClampSafetySen;
						fbClprClampChk(bEn := TRUE);
					END_IF

				END_IF

				IF fbClprClampChk.udiStatus = 0 AND fbEnt.udiStatus = 0 THEN
					eStatus		:= Done;

				ELSIF fbClprClampChk.udiStatus > 0 AND fbClprClampChk.udiStatus < 65534 THEN
					bClprClampCtrl		:= FALSE;

					eStatus			:= Error;

					IF fbClprClampChk.udiStatus = 1503 THEN
						udiStatus	:= 10034;	//Clamper Clamp Sensor On Time Out In Clamp Check While Conveyor Enter With Clamper
					ELSIF fbClprClampChk.udiStatus = 1506 THEN
						udiStatus	:= 10035;	//Clamper Unclamp Sensor Off Time Out In Clamp Check While Conveyor Enter With Clamper
					ELSIF fbClprClampChk.udiStatus = 1507 THEN
						udiStatus	:= 10036;	//Clamper Clamp Safety Sensor Error In Clamp Check While Conveyor Enter With Clamper
					ELSE
						udiStatus	:= fbClprClampChk.udiStatus;
					END_IF

				ELSIF fbEnt.udiStatus > 0 AND fbEnt.udiStatus < 65534 THEN
					eStatus		:= Error;

					IF fbEnt.udiStatus = 1101 THEN
						udiStatus	:= 10037;	//Transfer In Time Out While Entering Magazine
					ELSE
						udiStatus	:= fbEnt.udiStatus;
					END_IF

				END_IF

			END_IF

		MagConvActPreExit:
			IF eStatus = Idle OR eStatus = Busy THEN

				eStatus	:= Busy;

				//Conveyor Run
				fbPreExit.bConvLToR		:= (p_eDirection = ConvDirLToR) OR (p_eDirection = ConvDirRToR);
				fbPreExit.tTxDlyTm		:= DINT_TO_TIME(p_diInitTm);

				IF fbPreExit.bConvLToR = TRUE THEN
					fbPreExit.bEndSen	:= p_bRightSen;
				ELSE
					fbPreExit.bEndSen	:= p_bLeftSen;
				END_IF

				fbPreExit(bEn := TRUE);

				bMtrSigOnOrLToR	:= fbPreExit.bMtrSigOnOrLToR;
				bMtrDirOrRToL	:= fbPreExit.bMtrDirOrRToL;

				IF fbPreExit.udiStatus = 0 THEN
					IF fbPreExit.bEndSen = TRUE THEN
						eStatus	:= Done;
					ELSE
						udiStatus	:= 10046;	//Magazine Not Detected While Pre-Exiting Magazine
						eStatus		:= Error;
					END_IF
				ELSIF fbPreExit.udiStatus < 65534 THEN
					udiStatus	:= fbPreExit.udiStatus;
					eStatus		:= Error;
				END_IF

			END_IF

		MagConvActPreExitClpr:
			IF eStatus = Idle OR eStatus = Busy THEN

				eStatus	:= Busy;

				CASE usiStep OF
					0:
						bClprClampCtrl		:= FALSE;

						fbClprUnclampChk.bExtSen		:= p_bClprClampSen;
						fbClprUnclampChk.bRetSen		:= p_bClprUnclampSen;
						fbClprUnclampChk.bRetSafety		:= p_bClprUnclampSafetySen;
						fbClprUnclampChk(bEn := TRUE);

						IF fbClprUnclampChk.udiStatus = 0 THEN
							usiStep		:= 1;
						ELSIF fbClprUnclampChk.udiStatus < 65534 THEN
							bClprClampCtrl		:= TRUE;

							eStatus			:= Error;

							IF fbClprUnclampChk.udiStatus = 1504 THEN
								udiStatus	:= 10013;	//Clamper Clamp Sensor Off Time Out In Unclamp Check While Conveyor Exit With Clamper
							ELSIF fbClprUnclampChk.udiStatus = 1505 THEN
								udiStatus	:= 10014;	//Clamper Unclamp Sensor On Time Out In Unclamp Check While Conveyor Exit With Clamper
							ELSIF fbClprUnclampChk.udiStatus = 1508 THEN
								udiStatus	:= 10015;	//Clamper Unclamp Safety Sensor Error In Unclamp Check While Conveyor Exit With Clamper
							ELSE
								udiStatus	:= fbClprUnclampChk.udiStatus;
							END_IF
						END_IF

					1:
						//Conveyor Run
						fbPreExit.bConvLToR		:= (p_eDirection = ConvDirLToR) OR (p_eDirection = ConvDirRToR);
						fbPreExit.tTxDlyTm		:= DINT_TO_TIME(p_diInitTm);

						IF fbPreExit.bConvLToR = TRUE THEN
							fbPreExit.bEndSen	:= p_bRightSen;
						ELSE
							fbPreExit.bEndSen	:= p_bLeftSen;
						END_IF

						fbPreExit(bEn := TRUE);

						bMtrSigOnOrLToR	:= fbPreExit.bMtrSigOnOrLToR;
						bMtrDirOrRToL	:= fbPreExit.bMtrDirOrRToL;

						IF fbPreExit.udiStatus = 0 THEN
							IF fbPreExit.bEndSen = TRUE THEN
								eStatus	:= Done;
							ELSE
								udiStatus	:= 10046;	//Magazine Not Detected While Pre-Exiting Magazine
								eStatus		:= Error;
							END_IF
						ELSIF fbPreExit.udiStatus < 65534 THEN
							udiStatus	:= fbPreExit.udiStatus;
							eStatus		:= Error;
						END_IF

				END_CASE

			END_IF

		MagConvActExit:
			IF eStatus = Idle OR eStatus = Busy THEN

				eStatus	:= Busy;

				//Conveyor Run
				fbExit.bConvLToR	:= (p_eDirection = ConvDirLToR) OR (p_eDirection = ConvDirRToR);
				fbExit.tTimeOut		:= DINT_TO_TIME(p_diTxOutTimeOut);

				IF fbExit.bConvLToR = TRUE THEN
					fbExit.bEndSen	:= p_bRightSen;
				ELSE
					fbExit.bEndSen	:= p_bLeftSen;
				END_IF

				fbExit(bEn := TRUE);

				bMtrSigOnOrLToR	:= fbExit.bMtrSigOnOrLToR;
				bMtrDirOrRToL	:= fbExit.bMtrDirOrRToL;

				IF fbExit.udiStatus = 0 THEN
					bHvMag		:= FALSE;
					eStatus		:= Done;
				ELSIF fbExit.udiStatus < 65534 THEN
					eStatus		:= Error;

					IF fbExit.udiStatus = 1101 THEN
						udiStatus	:= 10030;	//Transfer Out Time Out While Exiting Magazine
					ELSE
						udiStatus	:= fbExit.udiStatus;
					END_IF
				END_IF

			END_IF

		MagConvActExit1:
			IF eStatus = Idle OR eStatus = Busy THEN

				eStatus	:= Busy;

				//Conveyor Run
				fbExit1.bConvLToR		:= (p_eDirection = ConvDirLToR) OR (p_eDirection = ConvDirRToR);
				fbExit1.tTimeOut		:= DINT_TO_TIME(p_diTxOutTimeOut);

				IF fbExit1.bConvLToR = TRUE THEN
					fbExit1.bEndSen	:= p_bRightSen;
				ELSE
					fbExit1.bEndSen	:= p_bLeftSen;
				END_IF

				fbExit1(bEn := TRUE);

				bMtrSigOnOrLToR	:= fbExit1.bMtrSigOnOrLToR;
				bMtrDirOrRToL	:= fbExit1.bMtrDirOrRToL;

				IF fbExit1.udiStatus = 0 THEN
					bHvMag		:= FALSE;
					eStatus		:= Done;
				ELSIF fbExit1.udiStatus < 65534 THEN
					eStatus		:= Error;

					IF fbExit1.udiStatus = 1101 THEN
						udiStatus	:= 10032;	//Transfer Out Time Out While Exiting Magazinie
					ELSE
						udiStatus	:= fbExit1.udiStatus;
					END_IF
				END_IF

			END_IF

		MagConvActExitClpr:
			IF eStatus = Idle OR eStatus = Busy THEN

				eStatus	:= Busy;

				CASE usiStep OF
					0:
						bClprClampCtrl		:= FALSE;

						fbClprUnclampChk.bExtSen		:= p_bClprClampSen;
						fbClprUnclampChk.bRetSen		:= p_bClprUnclampSen;
						fbClprUnclampChk.bRetSafety		:= p_bClprUnclampSafetySen;
						fbClprUnclampChk(bEn := TRUE);

						IF fbClprUnclampChk.udiStatus = 0 THEN
							usiStep		:= 1;
						ELSIF fbClprUnclampChk.udiStatus < 65534 THEN
							bClprClampCtrl		:= TRUE;

							eStatus			:= Error;

							IF fbClprUnclampChk.udiStatus = 1504 THEN
								udiStatus	:= 10013;	//Clamper Clamp Sensor Off Time Out In Unclamp Check While Conveyor Exit With Clamper
							ELSIF fbClprUnclampChk.udiStatus = 1505 THEN
								udiStatus	:= 10014;	//Clamper Unclamp Sensor On Time Out In Unclamp Check While Conveyor Exit With Clamper
							ELSIF fbClprUnclampChk.udiStatus = 1508 THEN
								udiStatus	:= 10015;	//Clamper Unclamp Safety Sensor Error In Unclamp Check While Conveyor Exit With Clamper
							ELSE
								udiStatus	:= fbClprUnclampChk.udiStatus;
							END_IF
						END_IF

					1:
						//Conveyor Run
						fbExit.bConvLToR	:= (p_eDirection = ConvDirLToR) OR (p_eDirection = ConvDirRToR);
						fbExit.tTimeOut		:= DINT_TO_TIME(p_diTxOutTimeOut);

						IF fbExit.bConvLToR = TRUE THEN
							fbExit.bEndSen	:= p_bRightSen;
						ELSE
							fbExit.bEndSen	:= p_bLeftSen;
						END_IF

						fbExit(bEn := TRUE);

						bMtrSigOnOrLToR	:= fbExit.bMtrSigOnOrLToR;
						bMtrDirOrRToL	:= fbExit.bMtrDirOrRToL;

						IF fbExit.udiStatus = 0 THEN
							bHvMag		:= FALSE;
							eStatus		:= Done;
						ELSIF fbExit.udiStatus < 65534 THEN
							eStatus		:= Error;

							IF fbExit.udiStatus = 1101 THEN
								udiStatus	:= 10031;	//Transfer Out Time Out While Conveyor Exit With Clamper
							ELSE
								udiStatus	:= fbExit.udiStatus;
							END_IF
						END_IF

				END_CASE

			END_IF

		MagConvActExit1Clpr:
			IF eStatus = Idle OR eStatus = Busy THEN

				eStatus	:= Busy;

				CASE usiStep OF
					0:
						bClprClampCtrl		:= FALSE;

						fbClprUnclampChk.bExtSen		:= p_bClprClampSen;
						fbClprUnclampChk.bRetSen		:= p_bClprUnclampSen;
						fbClprUnclampChk.bRetSafety		:= p_bClprUnclampSafetySen;
						fbClprUnclampChk(bEn := TRUE);

						IF fbClprUnclampChk.udiStatus = 0 THEN
							usiStep		:= 1;
						ELSIF fbClprUnclampChk.udiStatus < 65534 THEN
							bClprClampCtrl		:= TRUE;

							eStatus			:= Error;

							IF fbClprUnclampChk.udiStatus = 1504 THEN
								udiStatus	:= 10025;	//Clamper Clamp Sensor Off Time Out In Unclamp Check While Conveyor Exit With Clamper
							ELSIF fbClprUnclampChk.udiStatus = 1505 THEN
								udiStatus	:= 10026;	//Clamper Unclamp Sensor On Time Out In Unclamp Check While Conveyor Exit With Clamper
							ELSIF fbClprUnclampChk.udiStatus = 1508 THEN
								udiStatus	:= 10027;	//Clamper Unclamp Safety Sensor Error In Unclamp Check While Conveyor Exit With Clamper
							ELSE
								udiStatus	:= fbClprUnclampChk.udiStatus;
							END_IF
						END_IF

					1:
						//Conveyor Run
						fbExit1.bConvLToR		:= (p_eDirection = ConvDirLToR) OR (p_eDirection = ConvDirRToR);
						fbExit1.tTimeOut		:= DINT_TO_TIME(p_diTxOutTimeOut);

						IF fbExit1.bConvLToR = TRUE THEN
							fbExit1.bEndSen	:= p_bRightSen;
						ELSE
							fbExit1.bEndSen	:= p_bLeftSen;
						END_IF

						fbExit1(bEn := TRUE);

						bMtrSigOnOrLToR	:= fbExit1.bMtrSigOnOrLToR;
						bMtrDirOrRToL	:= fbExit1.bMtrDirOrRToL;

						IF fbExit1.udiStatus = 0 THEN
							bHvMag		:= FALSE;
							eStatus		:= Done;
						ELSIF fbExit1.udiStatus < 65534 THEN
							eStatus		:= Error;

							IF fbExit1.udiStatus = 1101 THEN
								udiStatus	:= 10033;	//Transfer Out Time Out While Conveyor Exit With Clamper
							ELSE
								udiStatus	:= fbExit1.udiStatus;
							END_IF
						END_IF

				END_CASE

			END_IF

		MagConvActClprSetAll:
			IF eStatus = Idle OR eStatus = Busy THEN

				eStatus	:= Busy;

				bMtrSigOnOrLToR	:= FALSE;
				bMtrDirOrRToL	:= FALSE;

				bClprClampCtrl		:= TRUE;

				eStatus		:= Done;

			END_IF

		MagConvActClprRstAll:
			IF eStatus = Idle OR eStatus = Busy THEN

				eStatus	:= Busy;

				bMtrSigOnOrLToR	:= FALSE;
				bMtrDirOrRToL	:= FALSE;

				bClprClampCtrl		:= FALSE;

				eStatus		:= Done;

			END_IF

		MagConvActClprSetClamp:
			IF eStatus = Idle OR eStatus = Busy THEN

				eStatus	:= Busy;

				bMtrSigOnOrLToR	:= FALSE;
				bMtrDirOrRToL	:= FALSE;

				bClprClampCtrl		:= TRUE;

				eStatus		:= Done;

			END_IF

		MagConvActClprSetUnclamp:
			IF eStatus = Idle OR eStatus = Busy THEN

				eStatus	:= Busy;

				bMtrSigOnOrLToR	:= FALSE;
				bMtrDirOrRToL	:= FALSE;

				bClprClampCtrl		:= FALSE;

				eStatus		:= Done;

			END_IF

		MagConvActClprClamp:
			IF eStatus = Idle OR eStatus = Busy THEN

				eStatus	:= Busy;

				bMtrSigOnOrLToR	:= FALSE;
				bMtrDirOrRToL	:= FALSE;

				bClprClampCtrl		:= TRUE;

				fbClprClampChk.bExtSen		:= p_bClprClampSen;
				fbClprClampChk.bRetSen		:= p_bClprUnclampSen;
				fbClprClampChk.bExtSafety	:= p_bClprClampSafetySen;
				fbClprClampChk(bEn := TRUE);

				IF fbClprClampChk.udiStatus = 0 THEN
					eStatus		:= Done;
				ELSIF fbClprClampChk.udiStatus < 65534 THEN
					bClprClampCtrl		:= FALSE;

					eStatus			:= Error;

					IF fbClprClampChk.udiStatus = 1503 THEN
						udiStatus	:= 10016;	//Clamper Clamp Sensor On Time Out In Clamp Check While Clamper Clamp
					ELSIF fbClprClampChk.udiStatus = 1506 THEN
						udiStatus	:= 10017;	//Clamper Unclamp Sensor Off Time Out In Clamp Check While Clamper Clamp
					ELSIF fbClprClampChk.udiStatus = 1507 THEN
						udiStatus	:= 10018;	//Clamper Clamp Safety Sensor Error In Clamp Check While Clamper Clamp
					ELSE
						udiStatus	:= fbClprClampChk.udiStatus;
					END_IF
				END_IF
			END_IF

		MagConvActClprUnclamp:
			IF eStatus = Idle OR eStatus = Busy THEN

				eStatus	:= Busy;

				bMtrSigOnOrLToR	:= FALSE;
				bMtrDirOrRToL	:= FALSE;

				bClprClampCtrl		:= FALSE;

				fbClprUnclampChk.bExtSen		:= p_bClprClampSen;
				fbClprUnclampChk.bRetSen		:= p_bClprUnclampSen;
				fbClprUnclampChk.bRetSafety		:= p_bClprUnclampSafetySen;
				fbClprUnclampChk(bEn := TRUE);

				IF fbClprUnclampChk.udiStatus = 0 THEN
					eStatus		:= Done;
				ELSIF fbClprUnclampChk.udiStatus < 65534 THEN
					bClprClampCtrl		:= TRUE;

					eStatus			:= Error;

					IF fbClprUnclampChk.udiStatus = 1504 THEN
						udiStatus	:= 10019;	//Clamper Clamp Sensor Off Time Out In Unclamp Check While Clamper Unclamp
					ELSIF fbClprUnclampChk.udiStatus = 1505 THEN
						udiStatus	:= 10020;	//Clamper Unclamp Sensor On Time Out In Unclamp Check While Clamper Unclamp
					ELSIF fbClprUnclampChk.udiStatus = 1508 THEN
						udiStatus	:= 10021;	//Clamper Unclamp Safety Sensor Error In Unclamp Check While Clamper Unclamp
					ELSE
						udiStatus	:= fbClprUnclampChk.udiStatus;
					END_IF
				END_IF

			END_IF

		MagConvActStop:
			IF eStatus = Idle OR eStatus = Busy THEN

				eStatus	:= Busy;

				//Conveyor Run
				fbStop(bEn := TRUE);

				bMtrSigOnOrLToR	:= fbStop.bMtrSigOnOrLToR;
				bMtrDirOrRToL	:= fbStop.bMtrDirOrRToL;

				IF fbStop.udiStatus = 0 THEN
					eStatus	:= Done;
				ELSIF fbStop.udiStatus < 65534 THEN
					udiStatus	:= fbStop.udiStatus;
					eStatus		:= Error;
				END_IF

			END_IF

		MagConvActStopClpr:
			IF eStatus = Idle OR eStatus = Busy THEN

				eStatus	:= Busy;

				//Conveyor Run
				fbStop(bEn := TRUE);

				bMtrSigOnOrLToR	:= fbStop.bMtrSigOnOrLToR;
				bMtrDirOrRToL	:= fbStop.bMtrDirOrRToL;

				bClprClampCtrl		:= FALSE;

				fbClprUnclampChk.bExtSen		:= p_bClprClampSen;
				fbClprUnclampChk.bRetSen		:= p_bClprUnclampSen;
				fbClprUnclampChk.bRetSafety		:= p_bClprUnclampSafetySen;
				fbClprUnclampChk(bEn := TRUE);

				IF fbStop.udiStatus = 0 AND fbClprUnclampChk.udiStatus = 0 THEN
					eStatus		:= Done;
				ELSIF fbStop.udiStatus > 0 AND fbStop.udiStatus < 65534 THEN
					udiStatus	:= fbStop.udiStatus;
					eStatus		:= Error;
				ELSIF fbClprUnclampChk.udiStatus > 0 AND fbClprUnclampChk.udiStatus < 65534 THEN
					bClprClampCtrl		:= TRUE;

					eStatus			:= Error;

					IF fbClprUnclampChk.udiStatus = 1504 THEN
						udiStatus	:= 10022;	//Clamper Clamp Sensor Off Time Out In Unclamp Check While Stop With Clamper
					ELSIF fbClprUnclampChk.udiStatus = 1505 THEN
						udiStatus	:= 10023;	//Clamper Unclamp Sensor On Time Out In Unclamp Check While Stop With Clamper
					ELSIF fbClprUnclampChk.udiStatus = 1508 THEN
						udiStatus	:= 10024;	//Clamper Unclamp Safety Sensor Error In Unclamp Check While Stop With Clamper
					ELSE
						udiStatus	:= fbClprUnclampChk.udiStatus;
					END_IF
				END_IF

			END_IF

		MagConvActSetMtrSigOnOrLToR:
			IF eStatus = Idle OR eStatus = Busy THEN

				bMtrSigOnOrLToR	:= TRUE;

				eStatus		:= Done;

			END_IF

		MagConvActSetMtrDirOrRToL:
			IF eStatus = Idle OR eStatus = Busy THEN

				bMtrDirOrRToL	:= TRUE;

				eStatus		:= Done;

			END_IF

		MagConvActRstMtrSigOnOrLToR:
			IF eStatus = Idle OR eStatus = Busy THEN

				bMtrSigOnOrLToR	:= FALSE;

				eStatus		:= Done;

			END_IF

		MagConvActRstMtrDirOrRToL:
			IF eStatus = Idle OR eStatus = Busy THEN

				bMtrDirOrRToL	:= FALSE;

				eStatus		:= Done;

			END_IF

		MagConvActSetMtrAll:
			IF eStatus = Idle OR eStatus = Busy THEN

				bMtrSigOnOrLToR	:= TRUE;
				bMtrDirOrRToL	:= TRUE;

				eStatus		:= Done;

			END_IF

		MagConvActRstMtrAll:
			IF eStatus = Idle OR eStatus = Busy THEN

				bMtrSigOnOrLToR	:= FALSE;
				bMtrDirOrRToL	:= FALSE;

				eStatus		:= Done;

			END_IF

	END_CASE

END_ACTION
```
